// TIA Portal V19 export
FUNCTION "UF" : Void   // FC12, LAD
{ S7_Optimized_Access := 'TRUE' }
// stored: SetENOAutomatically false
   VAR_TEMP   // added for the SCL form of the ladder/FBD networks
      _w1 : Bool;
      _w2 : Bool;
   END_VAR
BEGIN

REGION Network 1: ABFV-201 OPEN F/B
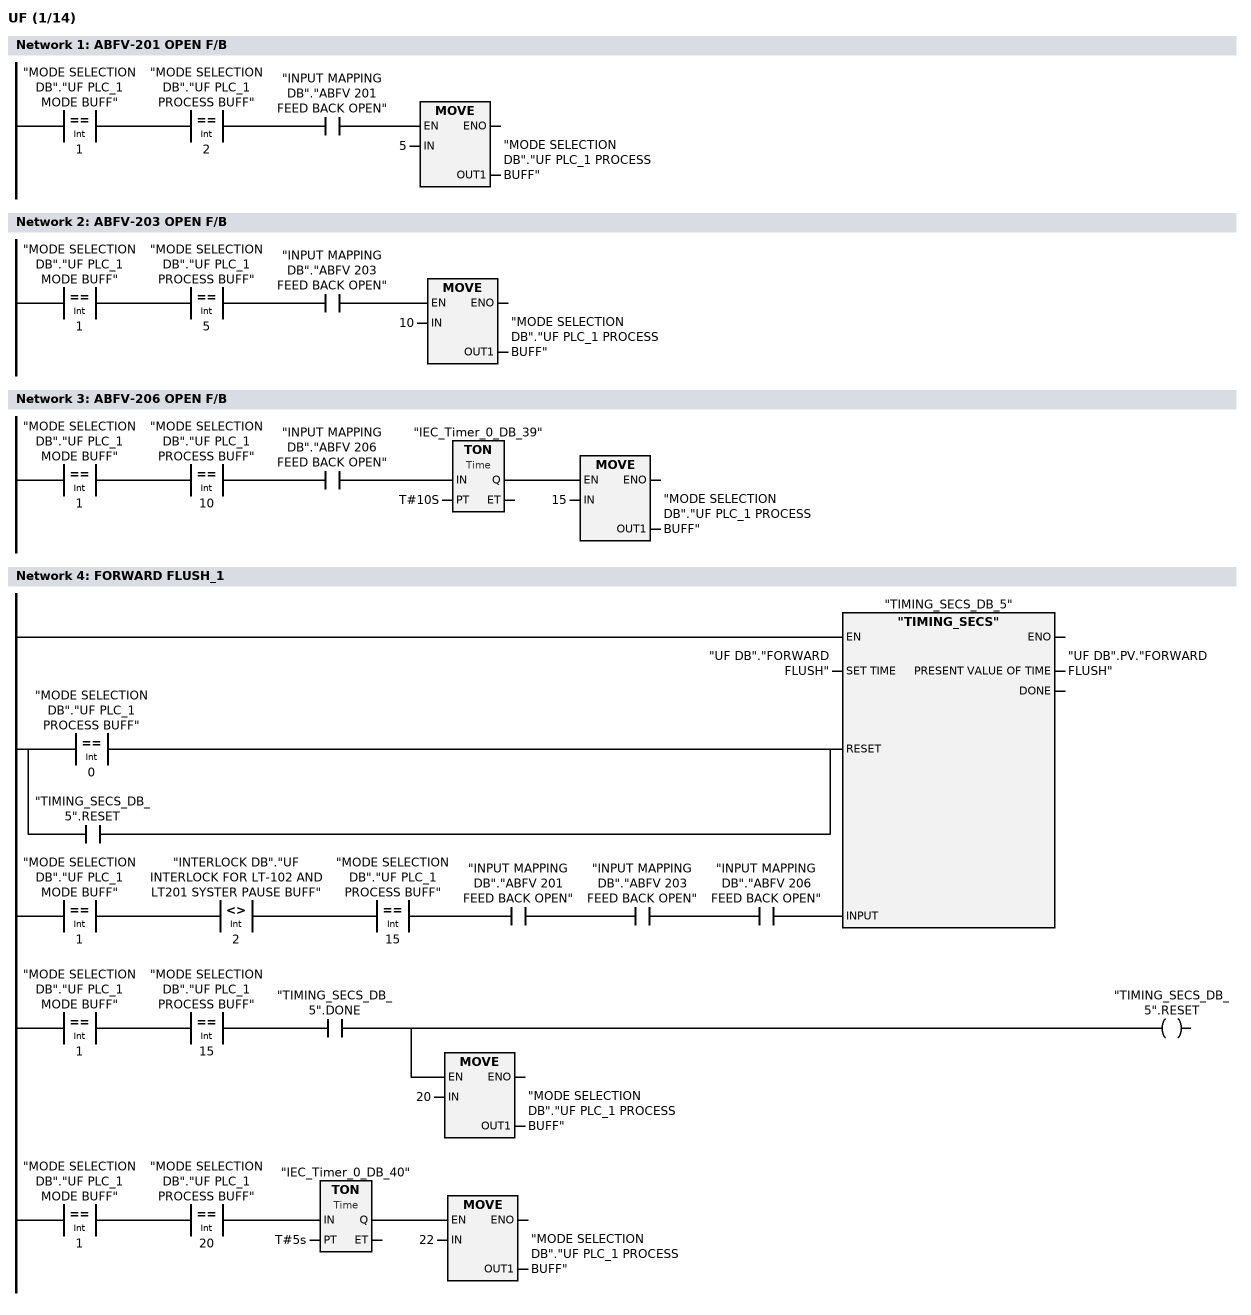
   RUNG wire#powerrail
      { S7_Templates := "SrcType := Int" } EQ_Contact(in1 := "MODE SELECTION DB"."UF PLC_1 MODE BUFF", in2 := 1)
      { S7_Templates := "SrcType := Int" } EQ_Contact(in1 := "MODE SELECTION DB"."UF PLC_1 PROCESS BUFF", in2 := 2)
      Contact( "INPUT MAPPING DB"."ABFV 201 FEED BACK OPEN" )
      Move(in := 5, out1 => "MODE SELECTION DB"."UF PLC_1 PROCESS BUFF")
   END_RUNG
   // the same network as SCL:
   IF ("MODE SELECTION DB"."UF PLC_1 MODE BUFF" = 1) AND ("MODE SELECTION DB"."UF PLC_1 PROCESS BUFF" = 2) AND "INPUT MAPPING DB"."ABFV 201 FEED BACK OPEN" THEN
       "MODE SELECTION DB"."UF PLC_1 PROCESS BUFF" := 5;
   END_IF;
END_REGION

REGION Network 2: ABFV-203 OPEN F/B
   RUNG wire#powerrail
      { S7_Templates := "SrcType := Int" } EQ_Contact(in1 := "MODE SELECTION DB"."UF PLC_1 MODE BUFF", in2 := 1)
      { S7_Templates := "SrcType := Int" } EQ_Contact(in1 := "MODE SELECTION DB"."UF PLC_1 PROCESS BUFF", in2 := 5)
      Contact( "INPUT MAPPING DB"."ABFV 203 FEED BACK OPEN" )
      Move(in := 10, out1 => "MODE SELECTION DB"."UF PLC_1 PROCESS BUFF")
   END_RUNG
   // the same network as SCL:
   IF ("MODE SELECTION DB"."UF PLC_1 MODE BUFF" = 1) AND ("MODE SELECTION DB"."UF PLC_1 PROCESS BUFF" = 5) AND "INPUT MAPPING DB"."ABFV 203 FEED BACK OPEN" THEN
       "MODE SELECTION DB"."UF PLC_1 PROCESS BUFF" := 10;
   END_IF;
END_REGION

REGION Network 3: ABFV-206 OPEN F/B
   RUNG wire#powerrail
      { S7_Templates := "SrcType := Int" } EQ_Contact(in1 := "MODE SELECTION DB"."UF PLC_1 MODE BUFF", in2 := 1)
      { S7_Templates := "SrcType := Int" } EQ_Contact(in1 := "MODE SELECTION DB"."UF PLC_1 PROCESS BUFF", in2 := 10)
      Contact( "INPUT MAPPING DB"."ABFV 206 FEED BACK OPEN" )
      { S7_Templates := "time_type := Time" } "IEC_Timer_0_DB_39".TON(pt := T#10S, et =>)
      Move(in := 15, out1 => "MODE SELECTION DB"."UF PLC_1 PROCESS BUFF")
   END_RUNG
   // the same network as SCL:
   "IEC_Timer_0_DB_39".TON(IN := ("MODE SELECTION DB"."UF PLC_1 MODE BUFF" = 1) AND ("MODE SELECTION DB"."UF PLC_1 PROCESS BUFF" = 10) AND "INPUT MAPPING DB"."ABFV 206 FEED BACK OPEN",
                           PT := T#10S);
   IF "IEC_Timer_0_DB_39".Q THEN "MODE SELECTION DB"."UF PLC_1 PROCESS BUFF" := 15; END_IF;
END_REGION

REGION Network 4: FORWARD FLUSH_1
   RUNG wire#powerrail
      "TIMING_SECS_DB_5"(RESET := wire#w1, INPUT := wire#w2, "SET TIME" := "UF DB"."FORWARD FLUSH", "PRESENT VALUE OF TIME" => "UF DB".PV."FORWARD FLUSH", DONE =>)
   END_RUNG
   RUNG wire#powerrail
      { S7_Templates := "SrcType := Int" } EQ_Contact(in1 := "MODE SELECTION DB"."UF PLC_1 PROCESS BUFF", in2 := 0)
   END_RUNG wire#w1
   RUNG wire#powerrail
      Contact( "TIMING_SECS_DB_5".RESET )
   END_RUNG wire#w1
   RUNG wire#powerrail
      { S7_Templates := "SrcType := Int" } EQ_Contact(in1 := "MODE SELECTION DB"."UF PLC_1 MODE BUFF", in2 := 1)
      { S7_Templates := "SrcType := Int" } NE_Contact(in1 := "INTERLOCK DB"."UF INTERLOCK FOR LT-102 AND LT201 SYSTER PAUSE BUFF", in2 := 2)
      { S7_Templates := "SrcType := Int" } EQ_Contact(in1 := "MODE SELECTION DB"."UF PLC_1 PROCESS BUFF", in2 := 15)
      Contact( "INPUT MAPPING DB"."ABFV 201 FEED BACK OPEN" )
      Contact( "INPUT MAPPING DB"."ABFV 203 FEED BACK OPEN" )
      Contact( "INPUT MAPPING DB"."ABFV 206 FEED BACK OPEN" )
   END_RUNG wire#w2
   RUNG wire#powerrail
      { S7_Templates := "SrcType := Int" } EQ_Contact(in1 := "MODE SELECTION DB"."UF PLC_1 MODE BUFF", in2 := 1)
      { S7_Templates := "SrcType := Int" } EQ_Contact(in1 := "MODE SELECTION DB"."UF PLC_1 PROCESS BUFF", in2 := 15)
      Contact( "TIMING_SECS_DB_5".DONE )
      wire#w3
      Coil( "TIMING_SECS_DB_5".RESET )
   END_RUNG
   RUNG wire#w3
      Move(in := 20, out1 => "MODE SELECTION DB"."UF PLC_1 PROCESS BUFF")
   END_RUNG
   RUNG wire#powerrail
      { S7_Templates := "SrcType := Int" } EQ_Contact(in1 := "MODE SELECTION DB"."UF PLC_1 MODE BUFF", in2 := 1)
      { S7_Templates := "SrcType := Int" } EQ_Contact(in1 := "MODE SELECTION DB"."UF PLC_1 PROCESS BUFF", in2 := 20)
      { S7_Templates := "time_type := Time" } "IEC_Timer_0_DB_40".TON(pt := T#5s, et =>)
      Move(in := 22, out1 => "MODE SELECTION DB"."UF PLC_1 PROCESS BUFF")
   END_RUNG
   // the same network as SCL:
   "TIMING_SECS_DB_5"("SET TIME" := "UF DB"."FORWARD FLUSH",   // "TIMING_SECS"
                      RESET := ("MODE SELECTION DB"."UF PLC_1 PROCESS BUFF" = 0) OR "TIMING_SECS_DB_5".RESET,
                      INPUT := ("MODE SELECTION DB"."UF PLC_1 MODE BUFF" = 1) AND ("INTERLOCK DB"."UF INTERLOCK FOR LT-102 AND LT201 SYSTER PAUSE BUFF" <> 2) AND ("MODE SELECTION DB"."UF PLC_1 PROCESS BUFF" = 15) AND "INPUT MAPPING DB"."ABFV 201 FEED BACK OPEN" AND "INPUT MAPPING DB"."ABFV 203 FEED BACK OPEN" AND "INPUT MAPPING DB"."ABFV 206 FEED BACK OPEN",
                      "PRESENT VALUE OF TIME" => "UF DB".PV."FORWARD FLUSH");
   "TIMING_SECS_DB_5".RESET := ("MODE SELECTION DB"."UF PLC_1 MODE BUFF" = 1) AND ("MODE SELECTION DB"."UF PLC_1 PROCESS BUFF" = 15) AND "TIMING_SECS_DB_5".DONE;
   IF "TIMING_SECS_DB_5".RESET THEN "MODE SELECTION DB"."UF PLC_1 PROCESS BUFF" := 20; END_IF;
   "IEC_Timer_0_DB_40".TON(IN := ("MODE SELECTION DB"."UF PLC_1 MODE BUFF" = 1) AND ("MODE SELECTION DB"."UF PLC_1 PROCESS BUFF" = 20),
                           PT := T#5s);
   IF "IEC_Timer_0_DB_40".Q THEN "MODE SELECTION DB"."UF PLC_1 PROCESS BUFF" := 22; END_IF;
END_REGION

REGION Network 5: OPEN ALL VALVE NEXT PROCESS
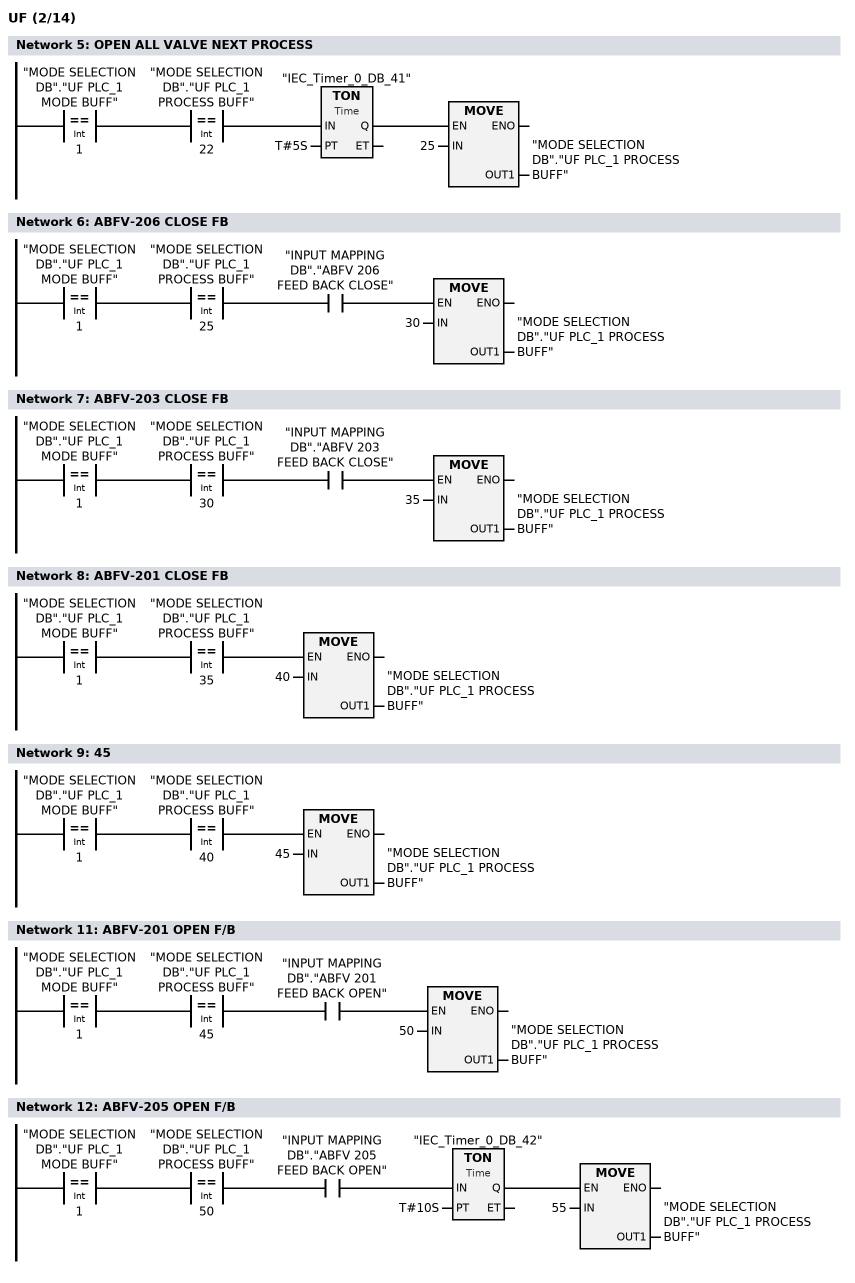
   RUNG wire#powerrail
      { S7_Templates := "SrcType := Int" } EQ_Contact(in1 := "MODE SELECTION DB"."UF PLC_1 MODE BUFF", in2 := 1)
      { S7_Templates := "SrcType := Int" } EQ_Contact(in1 := "MODE SELECTION DB"."UF PLC_1 PROCESS BUFF", in2 := 22)
      { S7_Templates := "time_type := Time" } "IEC_Timer_0_DB_41".TON(pt := T#5S, et =>)
      Move(in := 25, out1 => "MODE SELECTION DB"."UF PLC_1 PROCESS BUFF")
   END_RUNG
   // the same network as SCL:
   "IEC_Timer_0_DB_41".TON(IN := ("MODE SELECTION DB"."UF PLC_1 MODE BUFF" = 1) AND ("MODE SELECTION DB"."UF PLC_1 PROCESS BUFF" = 22),
                           PT := T#5S);
   IF "IEC_Timer_0_DB_41".Q THEN "MODE SELECTION DB"."UF PLC_1 PROCESS BUFF" := 25; END_IF;
END_REGION

REGION Network 6: ABFV-206 CLOSE FB
   RUNG wire#powerrail
      { S7_Templates := "SrcType := Int" } EQ_Contact(in1 := "MODE SELECTION DB"."UF PLC_1 MODE BUFF", in2 := 1)
      { S7_Templates := "SrcType := Int" } EQ_Contact(in1 := "MODE SELECTION DB"."UF PLC_1 PROCESS BUFF", in2 := 25)
      Contact( "INPUT MAPPING DB"."ABFV 206 FEED BACK CLOSE" )
      Move(in := 30, out1 => "MODE SELECTION DB"."UF PLC_1 PROCESS BUFF")
   END_RUNG
   // the same network as SCL:
   IF ("MODE SELECTION DB"."UF PLC_1 MODE BUFF" = 1) AND ("MODE SELECTION DB"."UF PLC_1 PROCESS BUFF" = 25) AND "INPUT MAPPING DB"."ABFV 206 FEED BACK CLOSE" THEN
       "MODE SELECTION DB"."UF PLC_1 PROCESS BUFF" := 30;
   END_IF;
END_REGION

REGION Network 7: ABFV-203 CLOSE FB
   RUNG wire#powerrail
      { S7_Templates := "SrcType := Int" } EQ_Contact(in1 := "MODE SELECTION DB"."UF PLC_1 MODE BUFF", in2 := 1)
      { S7_Templates := "SrcType := Int" } EQ_Contact(in1 := "MODE SELECTION DB"."UF PLC_1 PROCESS BUFF", in2 := 30)
      Contact( "INPUT MAPPING DB"."ABFV 203 FEED BACK CLOSE" )
      Move(in := 35, out1 => "MODE SELECTION DB"."UF PLC_1 PROCESS BUFF")
   END_RUNG
   // the same network as SCL:
   IF ("MODE SELECTION DB"."UF PLC_1 MODE BUFF" = 1) AND ("MODE SELECTION DB"."UF PLC_1 PROCESS BUFF" = 30) AND "INPUT MAPPING DB"."ABFV 203 FEED BACK CLOSE" THEN
       "MODE SELECTION DB"."UF PLC_1 PROCESS BUFF" := 35;
   END_IF;
END_REGION

REGION Network 8: ABFV-201 CLOSE FB
   RUNG wire#powerrail
      { S7_Templates := "SrcType := Int" } EQ_Contact(in1 := "MODE SELECTION DB"."UF PLC_1 MODE BUFF", in2 := 1)
      { S7_Templates := "SrcType := Int" } EQ_Contact(in1 := "MODE SELECTION DB"."UF PLC_1 PROCESS BUFF", in2 := 35)
      Move(in := 40, out1 => "MODE SELECTION DB"."UF PLC_1 PROCESS BUFF")
   END_RUNG
   // the same network as SCL:
   IF ("MODE SELECTION DB"."UF PLC_1 MODE BUFF" = 1) AND ("MODE SELECTION DB"."UF PLC_1 PROCESS BUFF" = 35) THEN
       "MODE SELECTION DB"."UF PLC_1 PROCESS BUFF" := 40;
   END_IF;
END_REGION

REGION Network 9: 45
   RUNG wire#powerrail
      { S7_Templates := "SrcType := Int" } EQ_Contact(in1 := "MODE SELECTION DB"."UF PLC_1 MODE BUFF", in2 := 1)
      { S7_Templates := "SrcType := Int" } EQ_Contact(in1 := "MODE SELECTION DB"."UF PLC_1 PROCESS BUFF", in2 := 40)
      Move(in := 45, out1 => "MODE SELECTION DB"."UF PLC_1 PROCESS BUFF")
   END_RUNG
   // the same network as SCL:
   IF ("MODE SELECTION DB"."UF PLC_1 MODE BUFF" = 1) AND ("MODE SELECTION DB"."UF PLC_1 PROCESS BUFF" = 40) THEN
       "MODE SELECTION DB"."UF PLC_1 PROCESS BUFF" := 45;
   END_IF;
END_REGION

REGION Network 11: ABFV-201 OPEN F/B
   RUNG wire#powerrail
      { S7_Templates := "SrcType := Int" } EQ_Contact(in1 := "MODE SELECTION DB"."UF PLC_1 MODE BUFF", in2 := 1)
      { S7_Templates := "SrcType := Int" } EQ_Contact(in1 := "MODE SELECTION DB"."UF PLC_1 PROCESS BUFF", in2 := 45)
      Contact( "INPUT MAPPING DB"."ABFV 201 FEED BACK OPEN" )
      Move(in := 50, out1 => "MODE SELECTION DB"."UF PLC_1 PROCESS BUFF")
   END_RUNG
   // the same network as SCL:
   IF ("MODE SELECTION DB"."UF PLC_1 MODE BUFF" = 1) AND ("MODE SELECTION DB"."UF PLC_1 PROCESS BUFF" = 45) AND "INPUT MAPPING DB"."ABFV 201 FEED BACK OPEN" THEN
       "MODE SELECTION DB"."UF PLC_1 PROCESS BUFF" := 50;
   END_IF;
END_REGION

REGION Network 12: ABFV-205 OPEN F/B
   RUNG wire#powerrail
      { S7_Templates := "SrcType := Int" } EQ_Contact(in1 := "MODE SELECTION DB"."UF PLC_1 MODE BUFF", in2 := 1)
      { S7_Templates := "SrcType := Int" } EQ_Contact(in1 := "MODE SELECTION DB"."UF PLC_1 PROCESS BUFF", in2 := 50)
      Contact( "INPUT MAPPING DB"."ABFV 205 FEED BACK OPEN" )
      { S7_Templates := "time_type := Time" } "IEC_Timer_0_DB_42".TON(pt := T#10S, et =>)
      Move(in := 55, out1 => "MODE SELECTION DB"."UF PLC_1 PROCESS BUFF")
   END_RUNG
   // the same network as SCL:
   "IEC_Timer_0_DB_42".TON(IN := ("MODE SELECTION DB"."UF PLC_1 MODE BUFF" = 1) AND ("MODE SELECTION DB"."UF PLC_1 PROCESS BUFF" = 50) AND "INPUT MAPPING DB"."ABFV 205 FEED BACK OPEN",
                           PT := T#10S);
   IF "IEC_Timer_0_DB_42".Q THEN "MODE SELECTION DB"."UF PLC_1 PROCESS BUFF" := 55; END_IF;
END_REGION

REGION Network 13: FILTRATION MODE
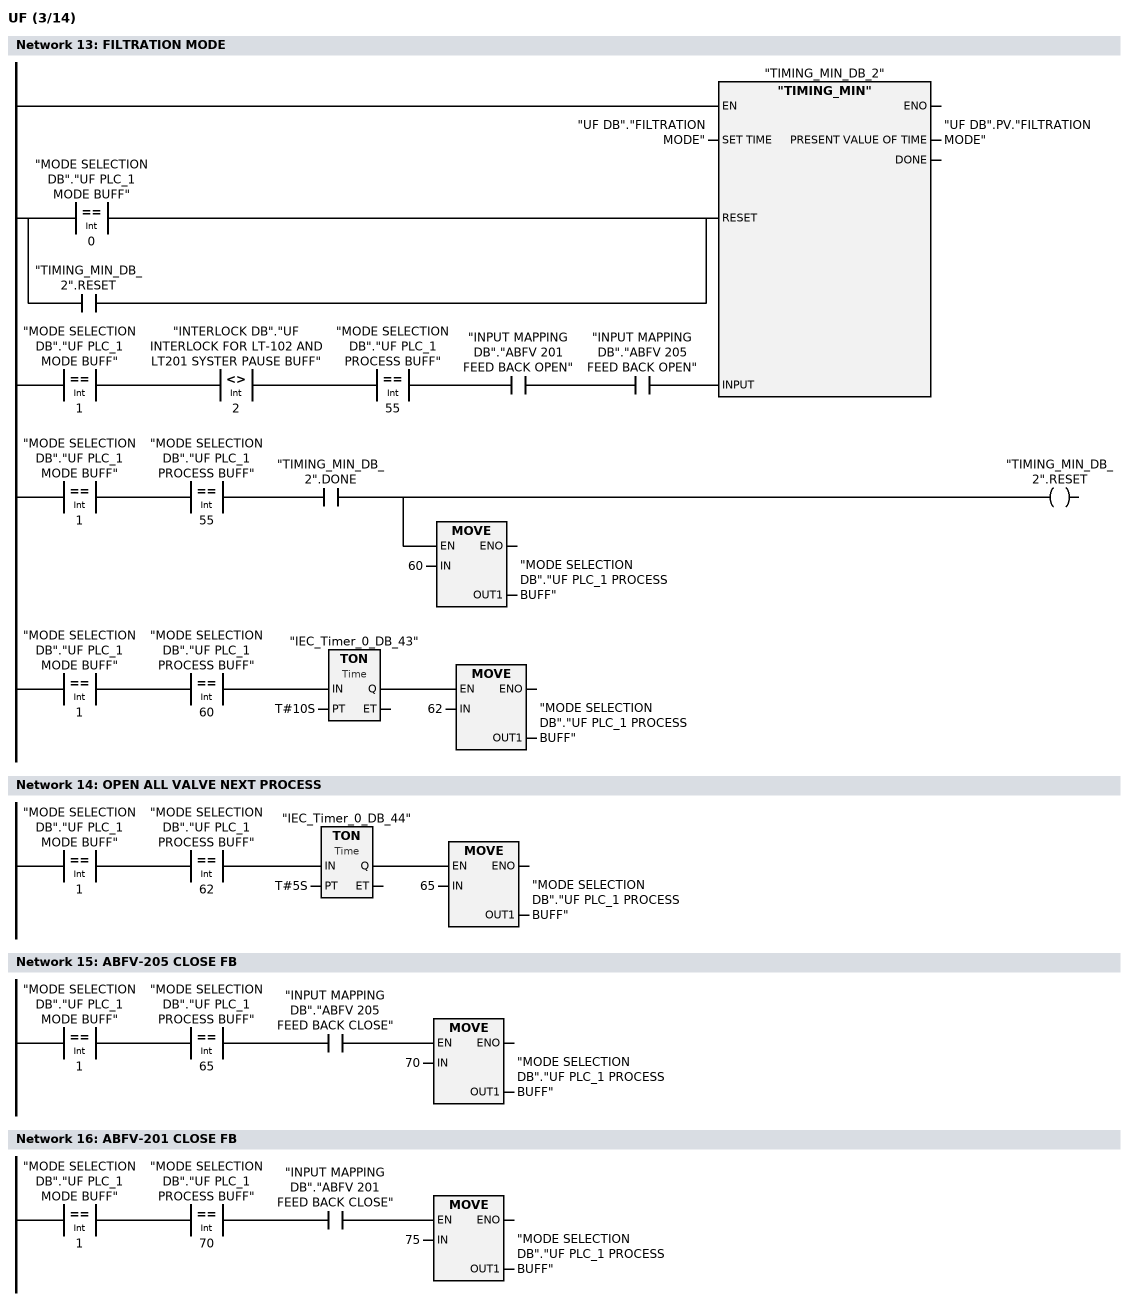
   RUNG wire#powerrail
      "TIMING_MIN_DB_2"(RESET := wire#w1, INPUT := wire#w2, "SET TIME" := "UF DB"."FILTRATION MODE", "PRESENT VALUE OF TIME" => "UF DB".PV."FILTRATION MODE", DONE =>)
   END_RUNG
   RUNG wire#powerrail
      { S7_Templates := "SrcType := Int" } EQ_Contact(in1 := "MODE SELECTION DB"."UF PLC_1 MODE BUFF", in2 := 0)
   END_RUNG wire#w1
   RUNG wire#powerrail
      Contact( "TIMING_MIN_DB_2".RESET )
   END_RUNG wire#w1
   RUNG wire#powerrail
      { S7_Templates := "SrcType := Int" } EQ_Contact(in1 := "MODE SELECTION DB"."UF PLC_1 MODE BUFF", in2 := 1)
      { S7_Templates := "SrcType := Int" } NE_Contact(in1 := "INTERLOCK DB"."UF INTERLOCK FOR LT-102 AND LT201 SYSTER PAUSE BUFF", in2 := 2)
      { S7_Templates := "SrcType := Int" } EQ_Contact(in1 := "MODE SELECTION DB"."UF PLC_1 PROCESS BUFF", in2 := 55)
      Contact( "INPUT MAPPING DB"."ABFV 201 FEED BACK OPEN" )
      Contact( "INPUT MAPPING DB"."ABFV 205 FEED BACK OPEN" )
   END_RUNG wire#w2
   RUNG wire#powerrail
      { S7_Templates := "SrcType := Int" } EQ_Contact(in1 := "MODE SELECTION DB"."UF PLC_1 MODE BUFF", in2 := 1)
      { S7_Templates := "SrcType := Int" } EQ_Contact(in1 := "MODE SELECTION DB"."UF PLC_1 PROCESS BUFF", in2 := 55)
      Contact( "TIMING_MIN_DB_2".DONE )
      wire#w3
      Coil( "TIMING_MIN_DB_2".RESET )
   END_RUNG
   RUNG wire#w3
      Move(in := 60, out1 => "MODE SELECTION DB"."UF PLC_1 PROCESS BUFF")
   END_RUNG
   RUNG wire#powerrail
      { S7_Templates := "SrcType := Int" } EQ_Contact(in1 := "MODE SELECTION DB"."UF PLC_1 MODE BUFF", in2 := 1)
      { S7_Templates := "SrcType := Int" } EQ_Contact(in1 := "MODE SELECTION DB"."UF PLC_1 PROCESS BUFF", in2 := 60)
      { S7_Templates := "time_type := Time" } "IEC_Timer_0_DB_43".TON(pt := T#10S, et =>)
      Move(in := 62, out1 => "MODE SELECTION DB"."UF PLC_1 PROCESS BUFF")
   END_RUNG
   // the same network as SCL:
   "TIMING_MIN_DB_2"("SET TIME" := "UF DB"."FILTRATION MODE",   // "TIMING_MIN"
                     RESET := ("MODE SELECTION DB"."UF PLC_1 MODE BUFF" = 0) OR "TIMING_MIN_DB_2".RESET,
                     INPUT := ("MODE SELECTION DB"."UF PLC_1 MODE BUFF" = 1) AND ("INTERLOCK DB"."UF INTERLOCK FOR LT-102 AND LT201 SYSTER PAUSE BUFF" <> 2) AND ("MODE SELECTION DB"."UF PLC_1 PROCESS BUFF" = 55) AND "INPUT MAPPING DB"."ABFV 201 FEED BACK OPEN" AND "INPUT MAPPING DB"."ABFV 205 FEED BACK OPEN",
                     "PRESENT VALUE OF TIME" => "UF DB".PV."FILTRATION MODE");
   "TIMING_MIN_DB_2".RESET := ("MODE SELECTION DB"."UF PLC_1 MODE BUFF" = 1) AND ("MODE SELECTION DB"."UF PLC_1 PROCESS BUFF" = 55) AND "TIMING_MIN_DB_2".DONE;
   IF "TIMING_MIN_DB_2".RESET THEN "MODE SELECTION DB"."UF PLC_1 PROCESS BUFF" := 60; END_IF;
   "IEC_Timer_0_DB_43".TON(IN := ("MODE SELECTION DB"."UF PLC_1 MODE BUFF" = 1) AND ("MODE SELECTION DB"."UF PLC_1 PROCESS BUFF" = 60),
                           PT := T#10S);
   IF "IEC_Timer_0_DB_43".Q THEN "MODE SELECTION DB"."UF PLC_1 PROCESS BUFF" := 62; END_IF;
END_REGION

REGION Network 14: OPEN ALL VALVE NEXT PROCESS
   RUNG wire#powerrail
      { S7_Templates := "SrcType := Int" } EQ_Contact(in1 := "MODE SELECTION DB"."UF PLC_1 MODE BUFF", in2 := 1)
      { S7_Templates := "SrcType := Int" } EQ_Contact(in1 := "MODE SELECTION DB"."UF PLC_1 PROCESS BUFF", in2 := 62)
      { S7_Templates := "time_type := Time" } "IEC_Timer_0_DB_44".TON(pt := T#5S, et =>)
      Move(in := 65, out1 => "MODE SELECTION DB"."UF PLC_1 PROCESS BUFF")
   END_RUNG
   // the same network as SCL:
   "IEC_Timer_0_DB_44".TON(IN := ("MODE SELECTION DB"."UF PLC_1 MODE BUFF" = 1) AND ("MODE SELECTION DB"."UF PLC_1 PROCESS BUFF" = 62),
                           PT := T#5S);
   IF "IEC_Timer_0_DB_44".Q THEN "MODE SELECTION DB"."UF PLC_1 PROCESS BUFF" := 65; END_IF;
END_REGION

REGION Network 15: ABFV-205 CLOSE FB
   RUNG wire#powerrail
      { S7_Templates := "SrcType := Int" } EQ_Contact(in1 := "MODE SELECTION DB"."UF PLC_1 MODE BUFF", in2 := 1)
      { S7_Templates := "SrcType := Int" } EQ_Contact(in1 := "MODE SELECTION DB"."UF PLC_1 PROCESS BUFF", in2 := 65)
      Contact( "INPUT MAPPING DB"."ABFV 205 FEED BACK CLOSE" )
      Move(in := 70, out1 => "MODE SELECTION DB"."UF PLC_1 PROCESS BUFF")
   END_RUNG
   // the same network as SCL:
   IF ("MODE SELECTION DB"."UF PLC_1 MODE BUFF" = 1) AND ("MODE SELECTION DB"."UF PLC_1 PROCESS BUFF" = 65) AND "INPUT MAPPING DB"."ABFV 205 FEED BACK CLOSE" THEN
       "MODE SELECTION DB"."UF PLC_1 PROCESS BUFF" := 70;
   END_IF;
END_REGION

REGION Network 16: ABFV-201 CLOSE FB
   RUNG wire#powerrail
      { S7_Templates := "SrcType := Int" } EQ_Contact(in1 := "MODE SELECTION DB"."UF PLC_1 MODE BUFF", in2 := 1)
      { S7_Templates := "SrcType := Int" } EQ_Contact(in1 := "MODE SELECTION DB"."UF PLC_1 PROCESS BUFF", in2 := 70)
      Contact( "INPUT MAPPING DB"."ABFV 201 FEED BACK CLOSE" )
      Move(in := 75, out1 => "MODE SELECTION DB"."UF PLC_1 PROCESS BUFF")
   END_RUNG
   // the same network as SCL:
   IF ("MODE SELECTION DB"."UF PLC_1 MODE BUFF" = 1) AND ("MODE SELECTION DB"."UF PLC_1 PROCESS BUFF" = 70) AND "INPUT MAPPING DB"."ABFV 201 FEED BACK CLOSE" THEN
       "MODE SELECTION DB"."UF PLC_1 PROCESS BUFF" := 75;
   END_IF;
END_REGION

REGION Network 17: 80
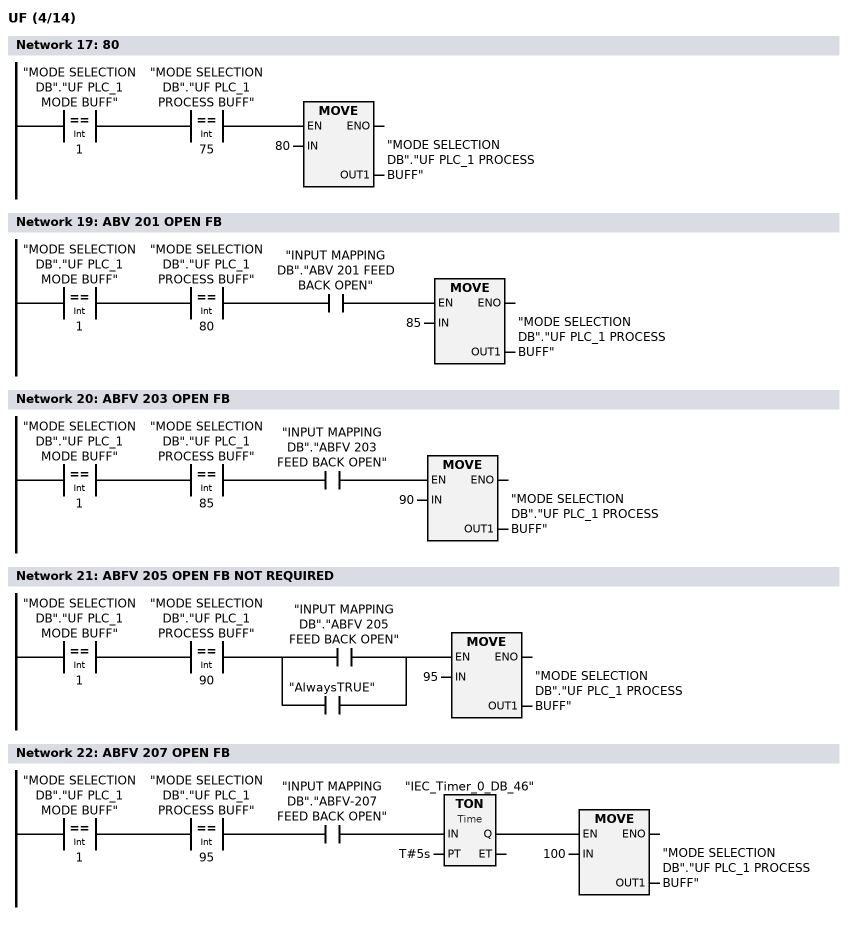
   RUNG wire#powerrail
      { S7_Templates := "SrcType := Int" } EQ_Contact(in1 := "MODE SELECTION DB"."UF PLC_1 MODE BUFF", in2 := 1)
      { S7_Templates := "SrcType := Int" } EQ_Contact(in1 := "MODE SELECTION DB"."UF PLC_1 PROCESS BUFF", in2 := 75)
      Move(in := 80, out1 => "MODE SELECTION DB"."UF PLC_1 PROCESS BUFF")
   END_RUNG
   // the same network as SCL:
   IF ("MODE SELECTION DB"."UF PLC_1 MODE BUFF" = 1) AND ("MODE SELECTION DB"."UF PLC_1 PROCESS BUFF" = 75) THEN
       "MODE SELECTION DB"."UF PLC_1 PROCESS BUFF" := 80;
   END_IF;
END_REGION

REGION Network 19: ABV 201 OPEN FB
   RUNG wire#powerrail
      { S7_Templates := "SrcType := Int" } EQ_Contact(in1 := "MODE SELECTION DB"."UF PLC_1 MODE BUFF", in2 := 1)
      { S7_Templates := "SrcType := Int" } EQ_Contact(in1 := "MODE SELECTION DB"."UF PLC_1 PROCESS BUFF", in2 := 80)
      Contact( "INPUT MAPPING DB"."ABV 201 FEED BACK OPEN" )
      Move(in := 85, out1 => "MODE SELECTION DB"."UF PLC_1 PROCESS BUFF")
   END_RUNG
   // the same network as SCL:
   IF ("MODE SELECTION DB"."UF PLC_1 MODE BUFF" = 1) AND ("MODE SELECTION DB"."UF PLC_1 PROCESS BUFF" = 80) AND "INPUT MAPPING DB"."ABV 201 FEED BACK OPEN" THEN
       "MODE SELECTION DB"."UF PLC_1 PROCESS BUFF" := 85;
   END_IF;
END_REGION

REGION Network 20: ABFV 203 OPEN FB
   RUNG wire#powerrail
      { S7_Templates := "SrcType := Int" } EQ_Contact(in1 := "MODE SELECTION DB"."UF PLC_1 MODE BUFF", in2 := 1)
      { S7_Templates := "SrcType := Int" } EQ_Contact(in1 := "MODE SELECTION DB"."UF PLC_1 PROCESS BUFF", in2 := 85)
      Contact( "INPUT MAPPING DB"."ABFV 203 FEED BACK OPEN" )
      Move(in := 90, out1 => "MODE SELECTION DB"."UF PLC_1 PROCESS BUFF")
   END_RUNG
   // the same network as SCL:
   IF ("MODE SELECTION DB"."UF PLC_1 MODE BUFF" = 1) AND ("MODE SELECTION DB"."UF PLC_1 PROCESS BUFF" = 85) AND "INPUT MAPPING DB"."ABFV 203 FEED BACK OPEN" THEN
       "MODE SELECTION DB"."UF PLC_1 PROCESS BUFF" := 90;
   END_IF;
END_REGION

REGION Network 21: ABFV 205 OPEN FB NOT REQUIRED
   RUNG wire#powerrail
      { S7_Templates := "SrcType := Int" } EQ_Contact(in1 := "MODE SELECTION DB"."UF PLC_1 MODE BUFF", in2 := 1)
      { S7_Templates := "SrcType := Int" } EQ_Contact(in1 := "MODE SELECTION DB"."UF PLC_1 PROCESS BUFF", in2 := 90)
      wire#w1
      Contact( "INPUT MAPPING DB"."ABFV 205 FEED BACK OPEN" )
      wire#w2
      Move(in := 95, out1 => "MODE SELECTION DB"."UF PLC_1 PROCESS BUFF")
   END_RUNG
   RUNG wire#w1
      Contact( "AlwaysTRUE" )
   END_RUNG wire#w2
   // the same network as SCL:
   IF ("MODE SELECTION DB"."UF PLC_1 MODE BUFF" = 1) AND ("MODE SELECTION DB"."UF PLC_1 PROCESS BUFF" = 90) AND ("INPUT MAPPING DB"."ABFV 205 FEED BACK OPEN" OR "AlwaysTRUE") THEN
       "MODE SELECTION DB"."UF PLC_1 PROCESS BUFF" := 95;
   END_IF;
END_REGION

REGION Network 22: ABFV 207 OPEN FB
   RUNG wire#powerrail
      { S7_Templates := "SrcType := Int" } EQ_Contact(in1 := "MODE SELECTION DB"."UF PLC_1 MODE BUFF", in2 := 1)
      { S7_Templates := "SrcType := Int" } EQ_Contact(in1 := "MODE SELECTION DB"."UF PLC_1 PROCESS BUFF", in2 := 95)
      Contact( "INPUT MAPPING DB"."ABFV-207 FEED BACK OPEN" )
      { S7_Templates := "time_type := Time" } "IEC_Timer_0_DB_46".TON(pt := T#5s, et =>)
      Move(in := 100, out1 => "MODE SELECTION DB"."UF PLC_1 PROCESS BUFF")
   END_RUNG
   // the same network as SCL:
   "IEC_Timer_0_DB_46".TON(IN := ("MODE SELECTION DB"."UF PLC_1 MODE BUFF" = 1) AND ("MODE SELECTION DB"."UF PLC_1 PROCESS BUFF" = 95) AND "INPUT MAPPING DB"."ABFV-207 FEED BACK OPEN",
                           PT := T#5s);
   IF "IEC_Timer_0_DB_46".Q THEN "MODE SELECTION DB"."UF PLC_1 PROCESS BUFF" := 100; END_IF;
END_REGION

REGION Network 23: AIR INLET
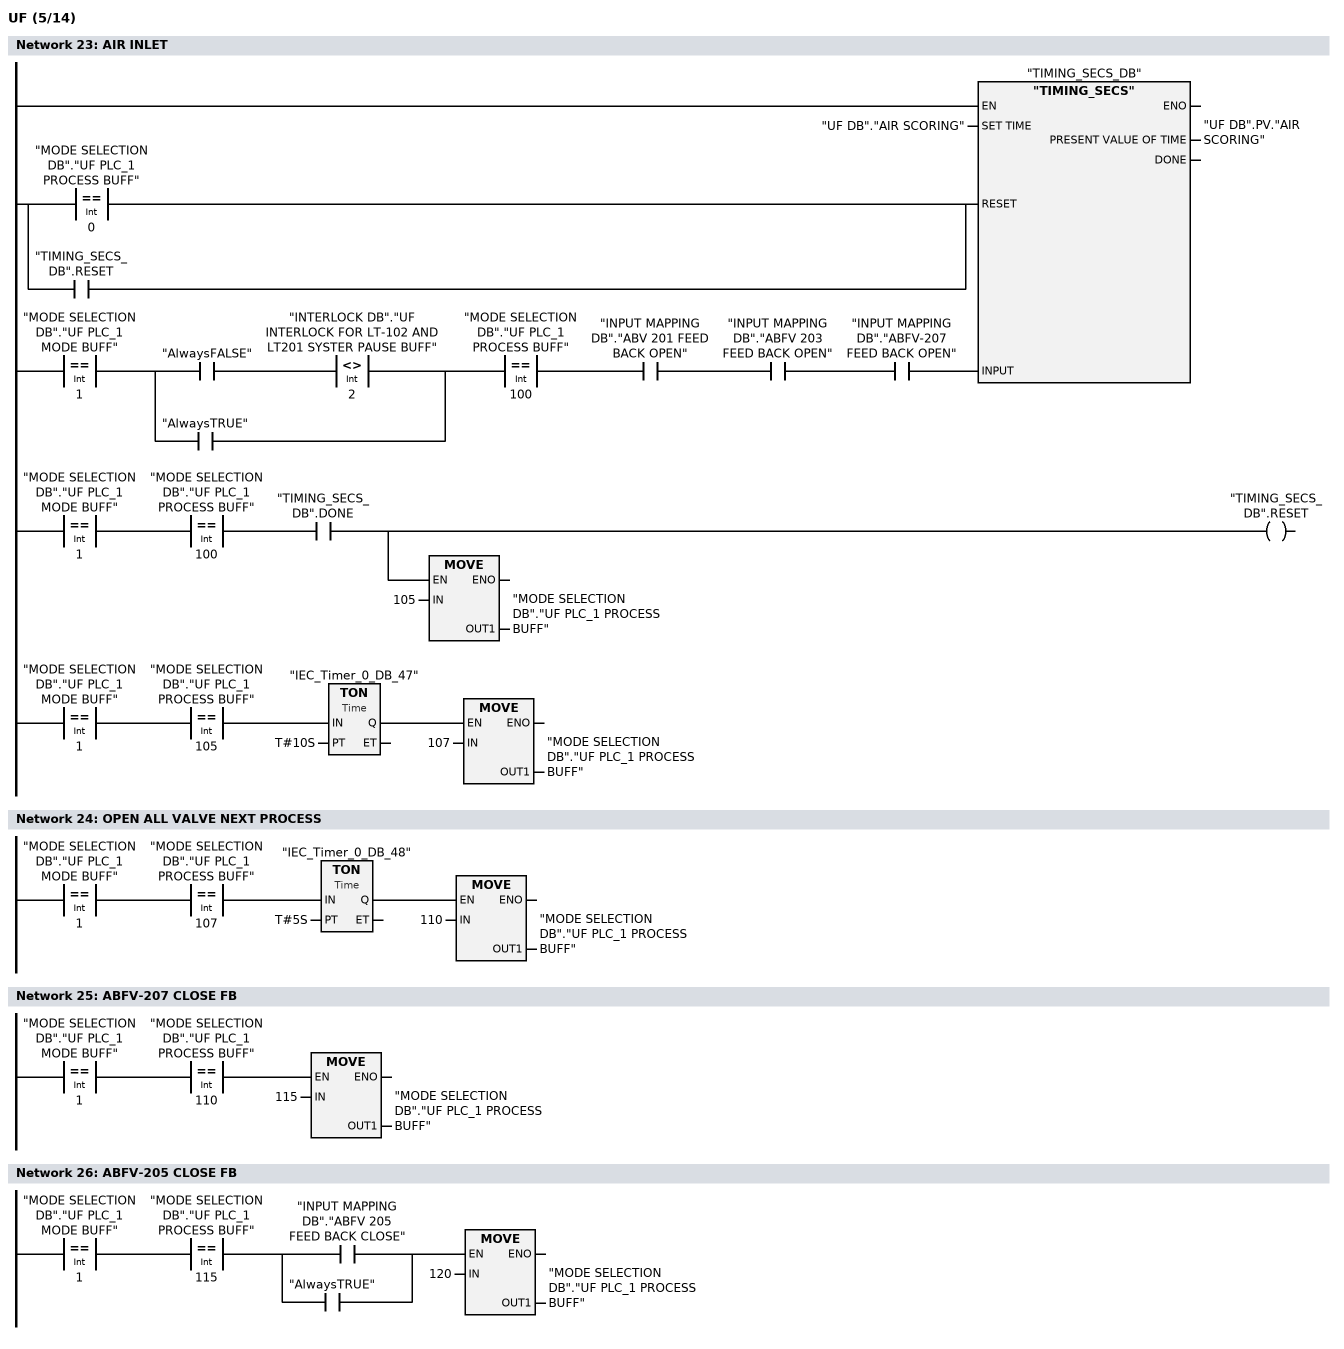
   RUNG wire#powerrail
      "TIMING_SECS_DB"(RESET := wire#w1, INPUT := wire#w4, "SET TIME" := "UF DB"."AIR SCORING", "PRESENT VALUE OF TIME" => "UF DB".PV."AIR SCORING", DONE =>)
   END_RUNG
   RUNG wire#powerrail
      { S7_Templates := "SrcType := Int" } EQ_Contact(in1 := "MODE SELECTION DB"."UF PLC_1 PROCESS BUFF", in2 := 0)
   END_RUNG wire#w1
   RUNG wire#powerrail
      Contact( "TIMING_SECS_DB".RESET )
   END_RUNG wire#w1
   RUNG wire#powerrail
      { S7_Templates := "SrcType := Int" } EQ_Contact(in1 := "MODE SELECTION DB"."UF PLC_1 MODE BUFF", in2 := 1)
      wire#w2
      Contact( "AlwaysFALSE" )
      { S7_Templates := "SrcType := Int" } NE_Contact(in1 := "INTERLOCK DB"."UF INTERLOCK FOR LT-102 AND LT201 SYSTER PAUSE BUFF", in2 := 2)
      wire#w3
      { S7_Templates := "SrcType := Int" } EQ_Contact(in1 := "MODE SELECTION DB"."UF PLC_1 PROCESS BUFF", in2 := 100)
      Contact( "INPUT MAPPING DB"."ABV 201 FEED BACK OPEN" )
      Contact( "INPUT MAPPING DB"."ABFV 203 FEED BACK OPEN" )
      Contact( "INPUT MAPPING DB"."ABFV-207 FEED BACK OPEN" )
   END_RUNG wire#w4
   RUNG wire#w2
      Contact( "AlwaysTRUE" )
   END_RUNG wire#w3
   RUNG wire#powerrail
      { S7_Templates := "SrcType := Int" } EQ_Contact(in1 := "MODE SELECTION DB"."UF PLC_1 MODE BUFF", in2 := 1)
      { S7_Templates := "SrcType := Int" } EQ_Contact(in1 := "MODE SELECTION DB"."UF PLC_1 PROCESS BUFF", in2 := 100)
      Contact( "TIMING_SECS_DB".DONE )
      wire#w5
      Coil( "TIMING_SECS_DB".RESET )
   END_RUNG
   RUNG wire#w5
      Move(in := 105, out1 => "MODE SELECTION DB"."UF PLC_1 PROCESS BUFF")
   END_RUNG
   RUNG wire#powerrail
      { S7_Templates := "SrcType := Int" } EQ_Contact(in1 := "MODE SELECTION DB"."UF PLC_1 MODE BUFF", in2 := 1)
      { S7_Templates := "SrcType := Int" } EQ_Contact(in1 := "MODE SELECTION DB"."UF PLC_1 PROCESS BUFF", in2 := 105)
      { S7_Templates := "time_type := Time" } "IEC_Timer_0_DB_47".TON(pt := T#10S, et =>)
      Move(in := 107, out1 => "MODE SELECTION DB"."UF PLC_1 PROCESS BUFF")
   END_RUNG
   // the same network as SCL:
   "TIMING_SECS_DB"("SET TIME" := "UF DB"."AIR SCORING",   // "TIMING_SECS"
                    RESET := ("MODE SELECTION DB"."UF PLC_1 PROCESS BUFF" = 0) OR "TIMING_SECS_DB".RESET,
                    INPUT := ("MODE SELECTION DB"."UF PLC_1 MODE BUFF" = 1) AND (("AlwaysFALSE" AND ("INTERLOCK DB"."UF INTERLOCK FOR LT-102 AND LT201 SYSTER PAUSE BUFF" <> 2)) OR "AlwaysTRUE") AND ("MODE SELECTION DB"."UF PLC_1 PROCESS BUFF" = 100) AND "INPUT MAPPING DB"."ABV 201 FEED BACK OPEN" AND "INPUT MAPPING DB"."ABFV 203 FEED BACK OPEN" AND "INPUT MAPPING DB"."ABFV-207 FEED BACK OPEN",
                    "PRESENT VALUE OF TIME" => "UF DB".PV."AIR SCORING");
   "TIMING_SECS_DB".RESET := ("MODE SELECTION DB"."UF PLC_1 MODE BUFF" = 1) AND ("MODE SELECTION DB"."UF PLC_1 PROCESS BUFF" = 100) AND "TIMING_SECS_DB".DONE;
   IF "TIMING_SECS_DB".RESET THEN "MODE SELECTION DB"."UF PLC_1 PROCESS BUFF" := 105; END_IF;
   "IEC_Timer_0_DB_47".TON(IN := ("MODE SELECTION DB"."UF PLC_1 MODE BUFF" = 1) AND ("MODE SELECTION DB"."UF PLC_1 PROCESS BUFF" = 105),
                           PT := T#10S);
   IF "IEC_Timer_0_DB_47".Q THEN "MODE SELECTION DB"."UF PLC_1 PROCESS BUFF" := 107; END_IF;
END_REGION

REGION Network 24: OPEN ALL VALVE NEXT PROCESS
   RUNG wire#powerrail
      { S7_Templates := "SrcType := Int" } EQ_Contact(in1 := "MODE SELECTION DB"."UF PLC_1 MODE BUFF", in2 := 1)
      { S7_Templates := "SrcType := Int" } EQ_Contact(in1 := "MODE SELECTION DB"."UF PLC_1 PROCESS BUFF", in2 := 107)
      { S7_Templates := "time_type := Time" } "IEC_Timer_0_DB_48".TON(pt := T#5S, et =>)
      Move(in := 110, out1 => "MODE SELECTION DB"."UF PLC_1 PROCESS BUFF")
   END_RUNG
   // the same network as SCL:
   "IEC_Timer_0_DB_48".TON(IN := ("MODE SELECTION DB"."UF PLC_1 MODE BUFF" = 1) AND ("MODE SELECTION DB"."UF PLC_1 PROCESS BUFF" = 107),
                           PT := T#5S);
   IF "IEC_Timer_0_DB_48".Q THEN "MODE SELECTION DB"."UF PLC_1 PROCESS BUFF" := 110; END_IF;
END_REGION

REGION Network 25: ABFV-207 CLOSE FB
   RUNG wire#powerrail
      { S7_Templates := "SrcType := Int" } EQ_Contact(in1 := "MODE SELECTION DB"."UF PLC_1 MODE BUFF", in2 := 1)
      { S7_Templates := "SrcType := Int" } EQ_Contact(in1 := "MODE SELECTION DB"."UF PLC_1 PROCESS BUFF", in2 := 110)
      Move(in := 115, out1 => "MODE SELECTION DB"."UF PLC_1 PROCESS BUFF")
   END_RUNG
   // the same network as SCL:
   IF ("MODE SELECTION DB"."UF PLC_1 MODE BUFF" = 1) AND ("MODE SELECTION DB"."UF PLC_1 PROCESS BUFF" = 110) THEN
       "MODE SELECTION DB"."UF PLC_1 PROCESS BUFF" := 115;
   END_IF;
END_REGION

REGION Network 26: ABFV-205 CLOSE FB
   RUNG wire#powerrail
      { S7_Templates := "SrcType := Int" } EQ_Contact(in1 := "MODE SELECTION DB"."UF PLC_1 MODE BUFF", in2 := 1)
      { S7_Templates := "SrcType := Int" } EQ_Contact(in1 := "MODE SELECTION DB"."UF PLC_1 PROCESS BUFF", in2 := 115)
      wire#w1
      Contact( "INPUT MAPPING DB"."ABFV 205 FEED BACK CLOSE" )
      wire#w2
      Move(in := 120, out1 => "MODE SELECTION DB"."UF PLC_1 PROCESS BUFF")
   END_RUNG
   RUNG wire#w1
      Contact( "AlwaysTRUE" )
   END_RUNG wire#w2
   // the same network as SCL:
   IF ("MODE SELECTION DB"."UF PLC_1 MODE BUFF" = 1) AND ("MODE SELECTION DB"."UF PLC_1 PROCESS BUFF" = 115) AND ("INPUT MAPPING DB"."ABFV 205 FEED BACK CLOSE" OR "AlwaysTRUE") THEN
       "MODE SELECTION DB"."UF PLC_1 PROCESS BUFF" := 120;
   END_IF;
END_REGION

REGION Network 27: ABFV-203 CLOSE FB
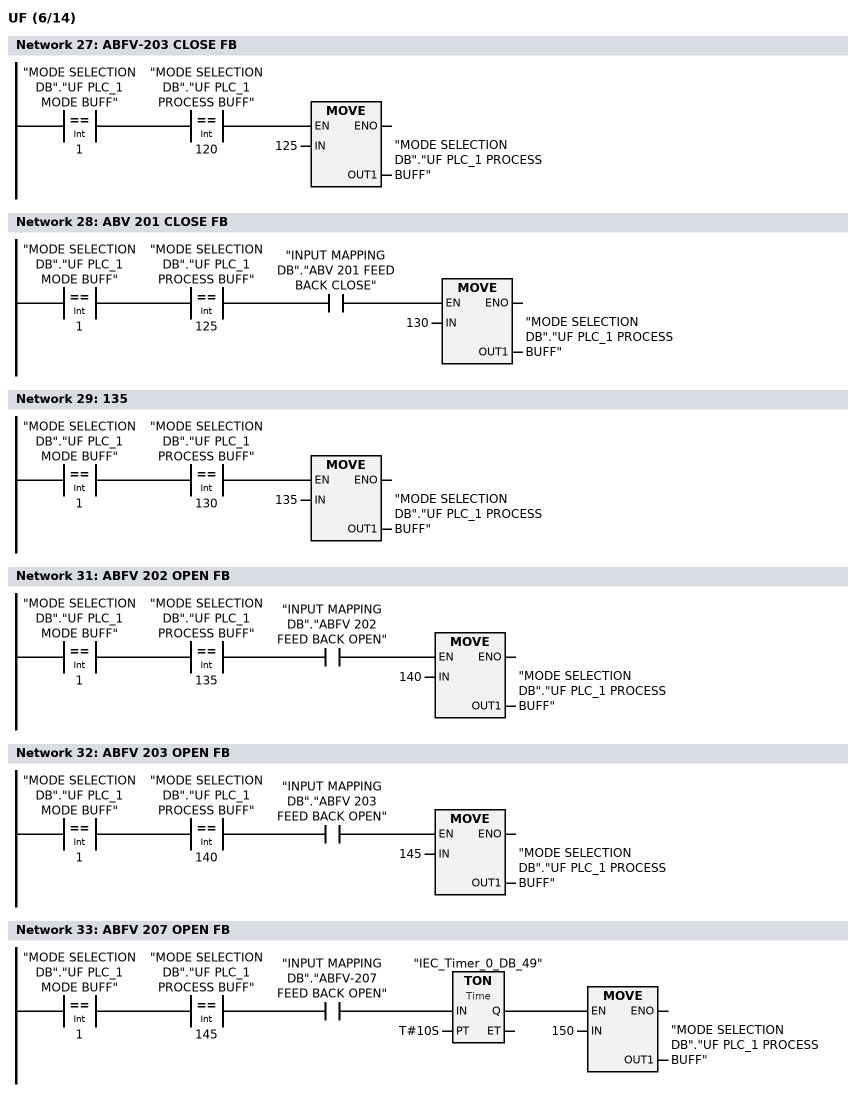
   RUNG wire#powerrail
      { S7_Templates := "SrcType := Int" } EQ_Contact(in1 := "MODE SELECTION DB"."UF PLC_1 MODE BUFF", in2 := 1)
      { S7_Templates := "SrcType := Int" } EQ_Contact(in1 := "MODE SELECTION DB"."UF PLC_1 PROCESS BUFF", in2 := 120)
      Move(in := 125, out1 => "MODE SELECTION DB"."UF PLC_1 PROCESS BUFF")
   END_RUNG
   // the same network as SCL:
   IF ("MODE SELECTION DB"."UF PLC_1 MODE BUFF" = 1) AND ("MODE SELECTION DB"."UF PLC_1 PROCESS BUFF" = 120) THEN
       "MODE SELECTION DB"."UF PLC_1 PROCESS BUFF" := 125;
   END_IF;
END_REGION

REGION Network 28: ABV 201 CLOSE FB
   RUNG wire#powerrail
      { S7_Templates := "SrcType := Int" } EQ_Contact(in1 := "MODE SELECTION DB"."UF PLC_1 MODE BUFF", in2 := 1)
      { S7_Templates := "SrcType := Int" } EQ_Contact(in1 := "MODE SELECTION DB"."UF PLC_1 PROCESS BUFF", in2 := 125)
      Contact( "INPUT MAPPING DB"."ABV 201 FEED BACK CLOSE" )
      Move(in := 130, out1 => "MODE SELECTION DB"."UF PLC_1 PROCESS BUFF")
   END_RUNG
   // the same network as SCL:
   IF ("MODE SELECTION DB"."UF PLC_1 MODE BUFF" = 1) AND ("MODE SELECTION DB"."UF PLC_1 PROCESS BUFF" = 125) AND "INPUT MAPPING DB"."ABV 201 FEED BACK CLOSE" THEN
       "MODE SELECTION DB"."UF PLC_1 PROCESS BUFF" := 130;
   END_IF;
END_REGION

REGION Network 29: 135
   RUNG wire#powerrail
      { S7_Templates := "SrcType := Int" } EQ_Contact(in1 := "MODE SELECTION DB"."UF PLC_1 MODE BUFF", in2 := 1)
      { S7_Templates := "SrcType := Int" } EQ_Contact(in1 := "MODE SELECTION DB"."UF PLC_1 PROCESS BUFF", in2 := 130)
      Move(in := 135, out1 => "MODE SELECTION DB"."UF PLC_1 PROCESS BUFF")
   END_RUNG
   // the same network as SCL:
   IF ("MODE SELECTION DB"."UF PLC_1 MODE BUFF" = 1) AND ("MODE SELECTION DB"."UF PLC_1 PROCESS BUFF" = 130) THEN
       "MODE SELECTION DB"."UF PLC_1 PROCESS BUFF" := 135;
   END_IF;
END_REGION

REGION Network 31: ABFV 202 OPEN FB
   RUNG wire#powerrail
      { S7_Templates := "SrcType := Int" } EQ_Contact(in1 := "MODE SELECTION DB"."UF PLC_1 MODE BUFF", in2 := 1)
      { S7_Templates := "SrcType := Int" } EQ_Contact(in1 := "MODE SELECTION DB"."UF PLC_1 PROCESS BUFF", in2 := 135)
      Contact( "INPUT MAPPING DB"."ABFV 202 FEED BACK OPEN" )
      Move(in := 140, out1 => "MODE SELECTION DB"."UF PLC_1 PROCESS BUFF")
   END_RUNG
   // the same network as SCL:
   IF ("MODE SELECTION DB"."UF PLC_1 MODE BUFF" = 1) AND ("MODE SELECTION DB"."UF PLC_1 PROCESS BUFF" = 135) AND "INPUT MAPPING DB"."ABFV 202 FEED BACK OPEN" THEN
       "MODE SELECTION DB"."UF PLC_1 PROCESS BUFF" := 140;
   END_IF;
END_REGION

REGION Network 32: ABFV 203 OPEN FB
   RUNG wire#powerrail
      { S7_Templates := "SrcType := Int" } EQ_Contact(in1 := "MODE SELECTION DB"."UF PLC_1 MODE BUFF", in2 := 1)
      { S7_Templates := "SrcType := Int" } EQ_Contact(in1 := "MODE SELECTION DB"."UF PLC_1 PROCESS BUFF", in2 := 140)
      Contact( "INPUT MAPPING DB"."ABFV 203 FEED BACK OPEN" )
      Move(in := 145, out1 => "MODE SELECTION DB"."UF PLC_1 PROCESS BUFF")
   END_RUNG
   // the same network as SCL:
   IF ("MODE SELECTION DB"."UF PLC_1 MODE BUFF" = 1) AND ("MODE SELECTION DB"."UF PLC_1 PROCESS BUFF" = 140) AND "INPUT MAPPING DB"."ABFV 203 FEED BACK OPEN" THEN
       "MODE SELECTION DB"."UF PLC_1 PROCESS BUFF" := 145;
   END_IF;
END_REGION

REGION Network 33: ABFV 207 OPEN FB
   RUNG wire#powerrail
      { S7_Templates := "SrcType := Int" } EQ_Contact(in1 := "MODE SELECTION DB"."UF PLC_1 MODE BUFF", in2 := 1)
      { S7_Templates := "SrcType := Int" } EQ_Contact(in1 := "MODE SELECTION DB"."UF PLC_1 PROCESS BUFF", in2 := 145)
      Contact( "INPUT MAPPING DB"."ABFV-207 FEED BACK OPEN" )
      { S7_Templates := "time_type := Time" } "IEC_Timer_0_DB_49".TON(pt := T#10S, et =>)
      Move(in := 150, out1 => "MODE SELECTION DB"."UF PLC_1 PROCESS BUFF")
   END_RUNG
   // the same network as SCL:
   "IEC_Timer_0_DB_49".TON(IN := ("MODE SELECTION DB"."UF PLC_1 MODE BUFF" = 1) AND ("MODE SELECTION DB"."UF PLC_1 PROCESS BUFF" = 145) AND "INPUT MAPPING DB"."ABFV-207 FEED BACK OPEN",
                           PT := T#10S);
   IF "IEC_Timer_0_DB_49".Q THEN "MODE SELECTION DB"."UF PLC_1 PROCESS BUFF" := 150; END_IF;
END_REGION

REGION Network 34: DAIN
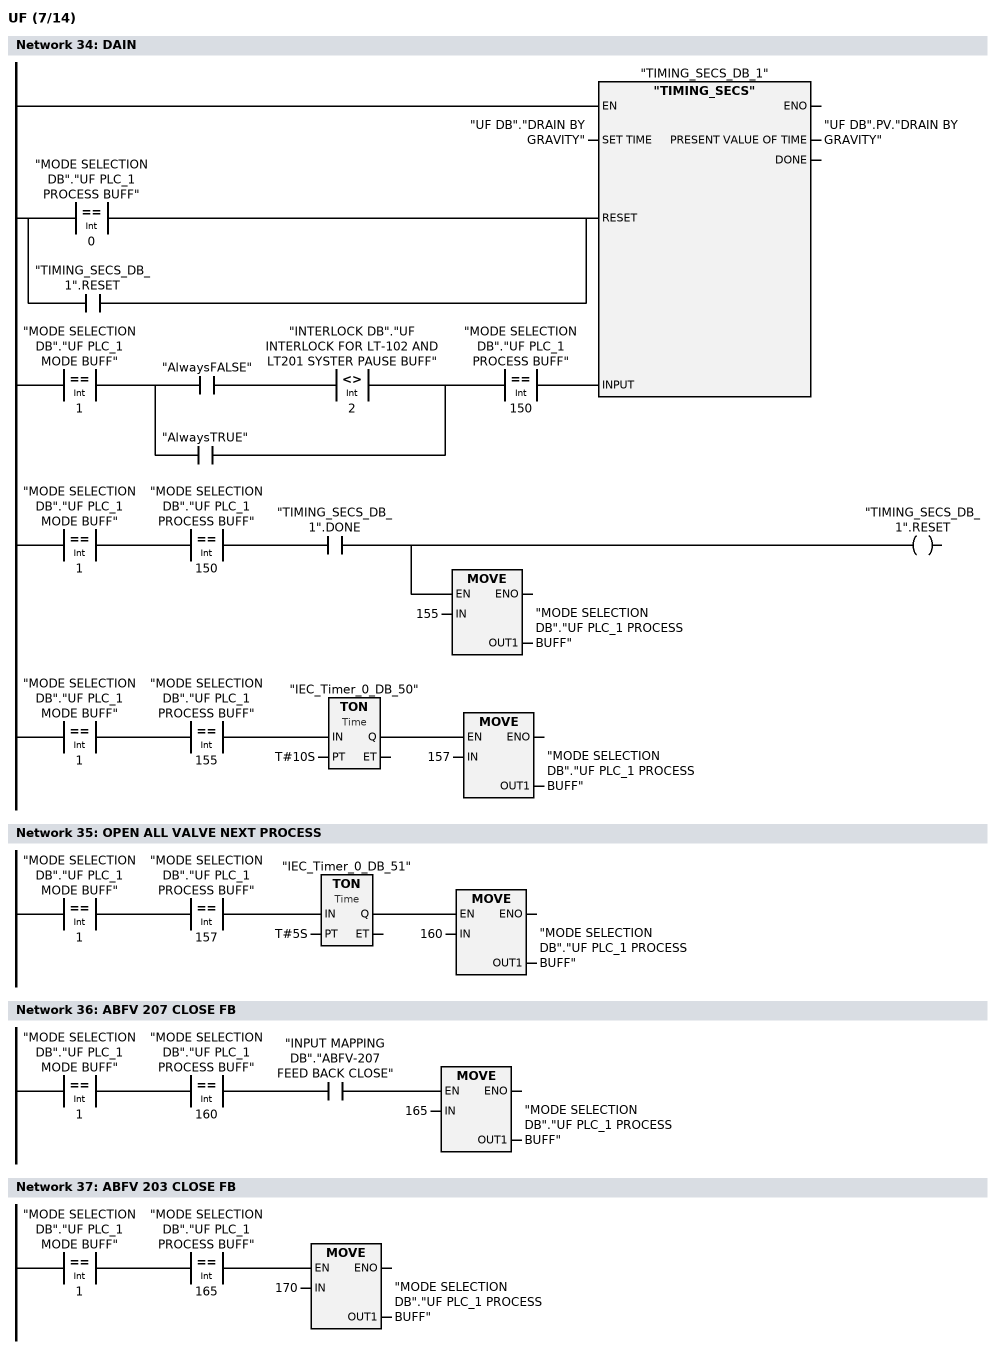
   RUNG wire#powerrail
      "TIMING_SECS_DB_1"(RESET := wire#w1, INPUT := wire#w4, "SET TIME" := "UF DB"."DRAIN BY GRAVITY", "PRESENT VALUE OF TIME" => "UF DB".PV."DRAIN BY GRAVITY", DONE =>)
   END_RUNG
   RUNG wire#powerrail
      { S7_Templates := "SrcType := Int" } EQ_Contact(in1 := "MODE SELECTION DB"."UF PLC_1 PROCESS BUFF", in2 := 0)
   END_RUNG wire#w1
   RUNG wire#powerrail
      Contact( "TIMING_SECS_DB_1".RESET )
   END_RUNG wire#w1
   RUNG wire#powerrail
      { S7_Templates := "SrcType := Int" } EQ_Contact(in1 := "MODE SELECTION DB"."UF PLC_1 MODE BUFF", in2 := 1)
      wire#w2
      Contact( "AlwaysFALSE" )
      { S7_Templates := "SrcType := Int" } NE_Contact(in1 := "INTERLOCK DB"."UF INTERLOCK FOR LT-102 AND LT201 SYSTER PAUSE BUFF", in2 := 2)
      wire#w3
      { S7_Templates := "SrcType := Int" } EQ_Contact(in1 := "MODE SELECTION DB"."UF PLC_1 PROCESS BUFF", in2 := 150)
   END_RUNG wire#w4
   RUNG wire#w2
      Contact( "AlwaysTRUE" )
   END_RUNG wire#w3
   RUNG wire#powerrail
      { S7_Templates := "SrcType := Int" } EQ_Contact(in1 := "MODE SELECTION DB"."UF PLC_1 MODE BUFF", in2 := 1)
      { S7_Templates := "SrcType := Int" } EQ_Contact(in1 := "MODE SELECTION DB"."UF PLC_1 PROCESS BUFF", in2 := 150)
      Contact( "TIMING_SECS_DB_1".DONE )
      wire#w5
      Coil( "TIMING_SECS_DB_1".RESET )
   END_RUNG
   RUNG wire#w5
      Move(in := 155, out1 => "MODE SELECTION DB"."UF PLC_1 PROCESS BUFF")
   END_RUNG
   RUNG wire#powerrail
      { S7_Templates := "SrcType := Int" } EQ_Contact(in1 := "MODE SELECTION DB"."UF PLC_1 MODE BUFF", in2 := 1)
      { S7_Templates := "SrcType := Int" } EQ_Contact(in1 := "MODE SELECTION DB"."UF PLC_1 PROCESS BUFF", in2 := 155)
      { S7_Templates := "time_type := Time" } "IEC_Timer_0_DB_50".TON(pt := T#10S, et =>)
      Move(in := 157, out1 => "MODE SELECTION DB"."UF PLC_1 PROCESS BUFF")
   END_RUNG
   // the same network as SCL:
   "TIMING_SECS_DB_1"("SET TIME" := "UF DB"."DRAIN BY GRAVITY",   // "TIMING_SECS"
                      RESET := ("MODE SELECTION DB"."UF PLC_1 PROCESS BUFF" = 0) OR "TIMING_SECS_DB_1".RESET,
                      INPUT := ("MODE SELECTION DB"."UF PLC_1 MODE BUFF" = 1) AND (("AlwaysFALSE" AND ("INTERLOCK DB"."UF INTERLOCK FOR LT-102 AND LT201 SYSTER PAUSE BUFF" <> 2)) OR "AlwaysTRUE") AND ("MODE SELECTION DB"."UF PLC_1 PROCESS BUFF" = 150),
                      "PRESENT VALUE OF TIME" => "UF DB".PV."DRAIN BY GRAVITY");
   "TIMING_SECS_DB_1".RESET := ("MODE SELECTION DB"."UF PLC_1 MODE BUFF" = 1) AND ("MODE SELECTION DB"."UF PLC_1 PROCESS BUFF" = 150) AND "TIMING_SECS_DB_1".DONE;
   IF "TIMING_SECS_DB_1".RESET THEN "MODE SELECTION DB"."UF PLC_1 PROCESS BUFF" := 155; END_IF;
   "IEC_Timer_0_DB_50".TON(IN := ("MODE SELECTION DB"."UF PLC_1 MODE BUFF" = 1) AND ("MODE SELECTION DB"."UF PLC_1 PROCESS BUFF" = 155),
                           PT := T#10S);
   IF "IEC_Timer_0_DB_50".Q THEN "MODE SELECTION DB"."UF PLC_1 PROCESS BUFF" := 157; END_IF;
END_REGION

REGION Network 35: OPEN ALL VALVE NEXT PROCESS
   RUNG wire#powerrail
      { S7_Templates := "SrcType := Int" } EQ_Contact(in1 := "MODE SELECTION DB"."UF PLC_1 MODE BUFF", in2 := 1)
      { S7_Templates := "SrcType := Int" } EQ_Contact(in1 := "MODE SELECTION DB"."UF PLC_1 PROCESS BUFF", in2 := 157)
      { S7_Templates := "time_type := Time" } "IEC_Timer_0_DB_51".TON(pt := T#5S, et =>)
      Move(in := 160, out1 => "MODE SELECTION DB"."UF PLC_1 PROCESS BUFF")
   END_RUNG
   // the same network as SCL:
   "IEC_Timer_0_DB_51".TON(IN := ("MODE SELECTION DB"."UF PLC_1 MODE BUFF" = 1) AND ("MODE SELECTION DB"."UF PLC_1 PROCESS BUFF" = 157),
                           PT := T#5S);
   IF "IEC_Timer_0_DB_51".Q THEN "MODE SELECTION DB"."UF PLC_1 PROCESS BUFF" := 160; END_IF;
END_REGION

REGION Network 36: ABFV 207 CLOSE FB
   RUNG wire#powerrail
      { S7_Templates := "SrcType := Int" } EQ_Contact(in1 := "MODE SELECTION DB"."UF PLC_1 MODE BUFF", in2 := 1)
      { S7_Templates := "SrcType := Int" } EQ_Contact(in1 := "MODE SELECTION DB"."UF PLC_1 PROCESS BUFF", in2 := 160)
      Contact( "INPUT MAPPING DB"."ABFV-207 FEED BACK CLOSE" )
      Move(in := 165, out1 => "MODE SELECTION DB"."UF PLC_1 PROCESS BUFF")
   END_RUNG
   // the same network as SCL:
   IF ("MODE SELECTION DB"."UF PLC_1 MODE BUFF" = 1) AND ("MODE SELECTION DB"."UF PLC_1 PROCESS BUFF" = 160) AND "INPUT MAPPING DB"."ABFV-207 FEED BACK CLOSE" THEN
       "MODE SELECTION DB"."UF PLC_1 PROCESS BUFF" := 165;
   END_IF;
END_REGION

REGION Network 37: ABFV 203 CLOSE FB
   RUNG wire#powerrail
      { S7_Templates := "SrcType := Int" } EQ_Contact(in1 := "MODE SELECTION DB"."UF PLC_1 MODE BUFF", in2 := 1)
      { S7_Templates := "SrcType := Int" } EQ_Contact(in1 := "MODE SELECTION DB"."UF PLC_1 PROCESS BUFF", in2 := 165)
      Move(in := 170, out1 => "MODE SELECTION DB"."UF PLC_1 PROCESS BUFF")
   END_RUNG
   // the same network as SCL:
   IF ("MODE SELECTION DB"."UF PLC_1 MODE BUFF" = 1) AND ("MODE SELECTION DB"."UF PLC_1 PROCESS BUFF" = 165) THEN
       "MODE SELECTION DB"."UF PLC_1 PROCESS BUFF" := 170;
   END_IF;
END_REGION

REGION Network 38: ABFV 202 CLOSE FB
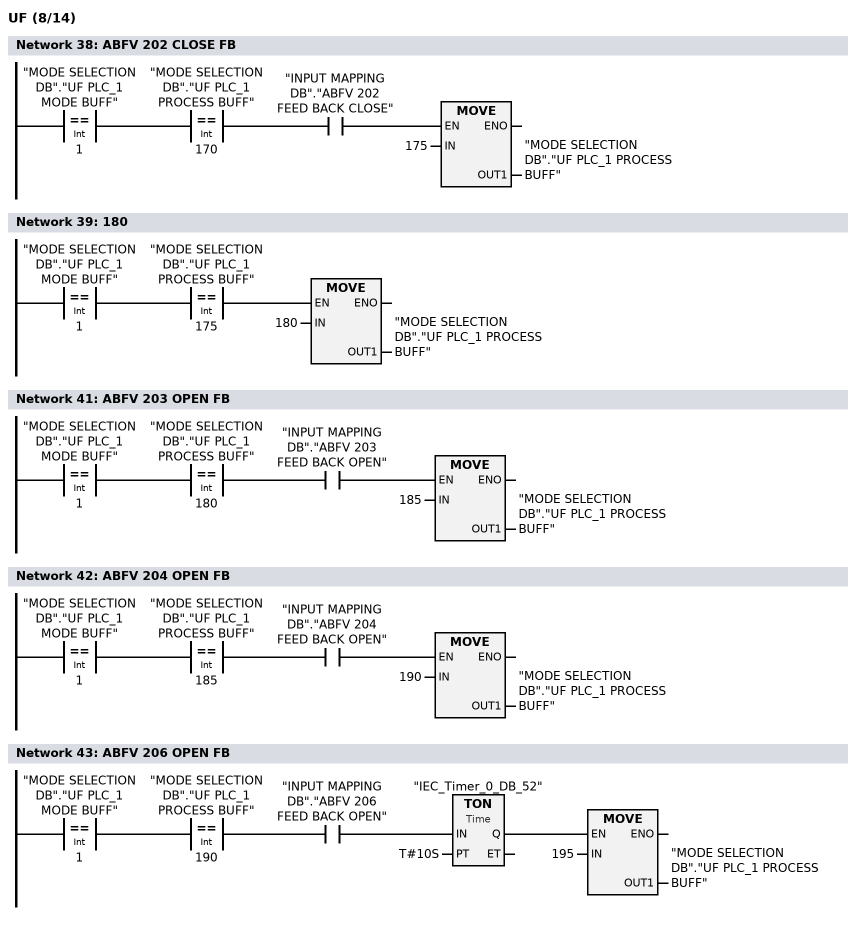
   RUNG wire#powerrail
      { S7_Templates := "SrcType := Int" } EQ_Contact(in1 := "MODE SELECTION DB"."UF PLC_1 MODE BUFF", in2 := 1)
      { S7_Templates := "SrcType := Int" } EQ_Contact(in1 := "MODE SELECTION DB"."UF PLC_1 PROCESS BUFF", in2 := 170)
      Contact( "INPUT MAPPING DB"."ABFV 202 FEED BACK CLOSE" )
      Move(in := 175, out1 => "MODE SELECTION DB"."UF PLC_1 PROCESS BUFF")
   END_RUNG
   // the same network as SCL:
   IF ("MODE SELECTION DB"."UF PLC_1 MODE BUFF" = 1) AND ("MODE SELECTION DB"."UF PLC_1 PROCESS BUFF" = 170) AND "INPUT MAPPING DB"."ABFV 202 FEED BACK CLOSE" THEN
       "MODE SELECTION DB"."UF PLC_1 PROCESS BUFF" := 175;
   END_IF;
END_REGION

REGION Network 39: 180
   RUNG wire#powerrail
      { S7_Templates := "SrcType := Int" } EQ_Contact(in1 := "MODE SELECTION DB"."UF PLC_1 MODE BUFF", in2 := 1)
      { S7_Templates := "SrcType := Int" } EQ_Contact(in1 := "MODE SELECTION DB"."UF PLC_1 PROCESS BUFF", in2 := 175)
      Move(in := 180, out1 => "MODE SELECTION DB"."UF PLC_1 PROCESS BUFF")
   END_RUNG
   // the same network as SCL:
   IF ("MODE SELECTION DB"."UF PLC_1 MODE BUFF" = 1) AND ("MODE SELECTION DB"."UF PLC_1 PROCESS BUFF" = 175) THEN
       "MODE SELECTION DB"."UF PLC_1 PROCESS BUFF" := 180;
   END_IF;
END_REGION

REGION Network 41: ABFV 203 OPEN FB
   RUNG wire#powerrail
      { S7_Templates := "SrcType := Int" } EQ_Contact(in1 := "MODE SELECTION DB"."UF PLC_1 MODE BUFF", in2 := 1)
      { S7_Templates := "SrcType := Int" } EQ_Contact(in1 := "MODE SELECTION DB"."UF PLC_1 PROCESS BUFF", in2 := 180)
      Contact( "INPUT MAPPING DB"."ABFV 203 FEED BACK OPEN" )
      Move(in := 185, out1 => "MODE SELECTION DB"."UF PLC_1 PROCESS BUFF")
   END_RUNG
   // the same network as SCL:
   IF ("MODE SELECTION DB"."UF PLC_1 MODE BUFF" = 1) AND ("MODE SELECTION DB"."UF PLC_1 PROCESS BUFF" = 180) AND "INPUT MAPPING DB"."ABFV 203 FEED BACK OPEN" THEN
       "MODE SELECTION DB"."UF PLC_1 PROCESS BUFF" := 185;
   END_IF;
END_REGION

REGION Network 42: ABFV 204 OPEN FB
   RUNG wire#powerrail
      { S7_Templates := "SrcType := Int" } EQ_Contact(in1 := "MODE SELECTION DB"."UF PLC_1 MODE BUFF", in2 := 1)
      { S7_Templates := "SrcType := Int" } EQ_Contact(in1 := "MODE SELECTION DB"."UF PLC_1 PROCESS BUFF", in2 := 185)
      Contact( "INPUT MAPPING DB"."ABFV 204 FEED BACK OPEN" )
      Move(in := 190, out1 => "MODE SELECTION DB"."UF PLC_1 PROCESS BUFF")
   END_RUNG
   // the same network as SCL:
   IF ("MODE SELECTION DB"."UF PLC_1 MODE BUFF" = 1) AND ("MODE SELECTION DB"."UF PLC_1 PROCESS BUFF" = 185) AND "INPUT MAPPING DB"."ABFV 204 FEED BACK OPEN" THEN
       "MODE SELECTION DB"."UF PLC_1 PROCESS BUFF" := 190;
   END_IF;
END_REGION

REGION Network 43: ABFV 206 OPEN FB
   RUNG wire#powerrail
      { S7_Templates := "SrcType := Int" } EQ_Contact(in1 := "MODE SELECTION DB"."UF PLC_1 MODE BUFF", in2 := 1)
      { S7_Templates := "SrcType := Int" } EQ_Contact(in1 := "MODE SELECTION DB"."UF PLC_1 PROCESS BUFF", in2 := 190)
      Contact( "INPUT MAPPING DB"."ABFV 206 FEED BACK OPEN" )
      { S7_Templates := "time_type := Time" } "IEC_Timer_0_DB_52".TON(pt := T#10S, et =>)
      Move(in := 195, out1 => "MODE SELECTION DB"."UF PLC_1 PROCESS BUFF")
   END_RUNG
   // the same network as SCL:
   "IEC_Timer_0_DB_52".TON(IN := ("MODE SELECTION DB"."UF PLC_1 MODE BUFF" = 1) AND ("MODE SELECTION DB"."UF PLC_1 PROCESS BUFF" = 190) AND "INPUT MAPPING DB"."ABFV 206 FEED BACK OPEN",
                           PT := T#10S);
   IF "IEC_Timer_0_DB_52".Q THEN "MODE SELECTION DB"."UF PLC_1 PROCESS BUFF" := 195; END_IF;
END_REGION

REGION Network 44: BACKWASH-1
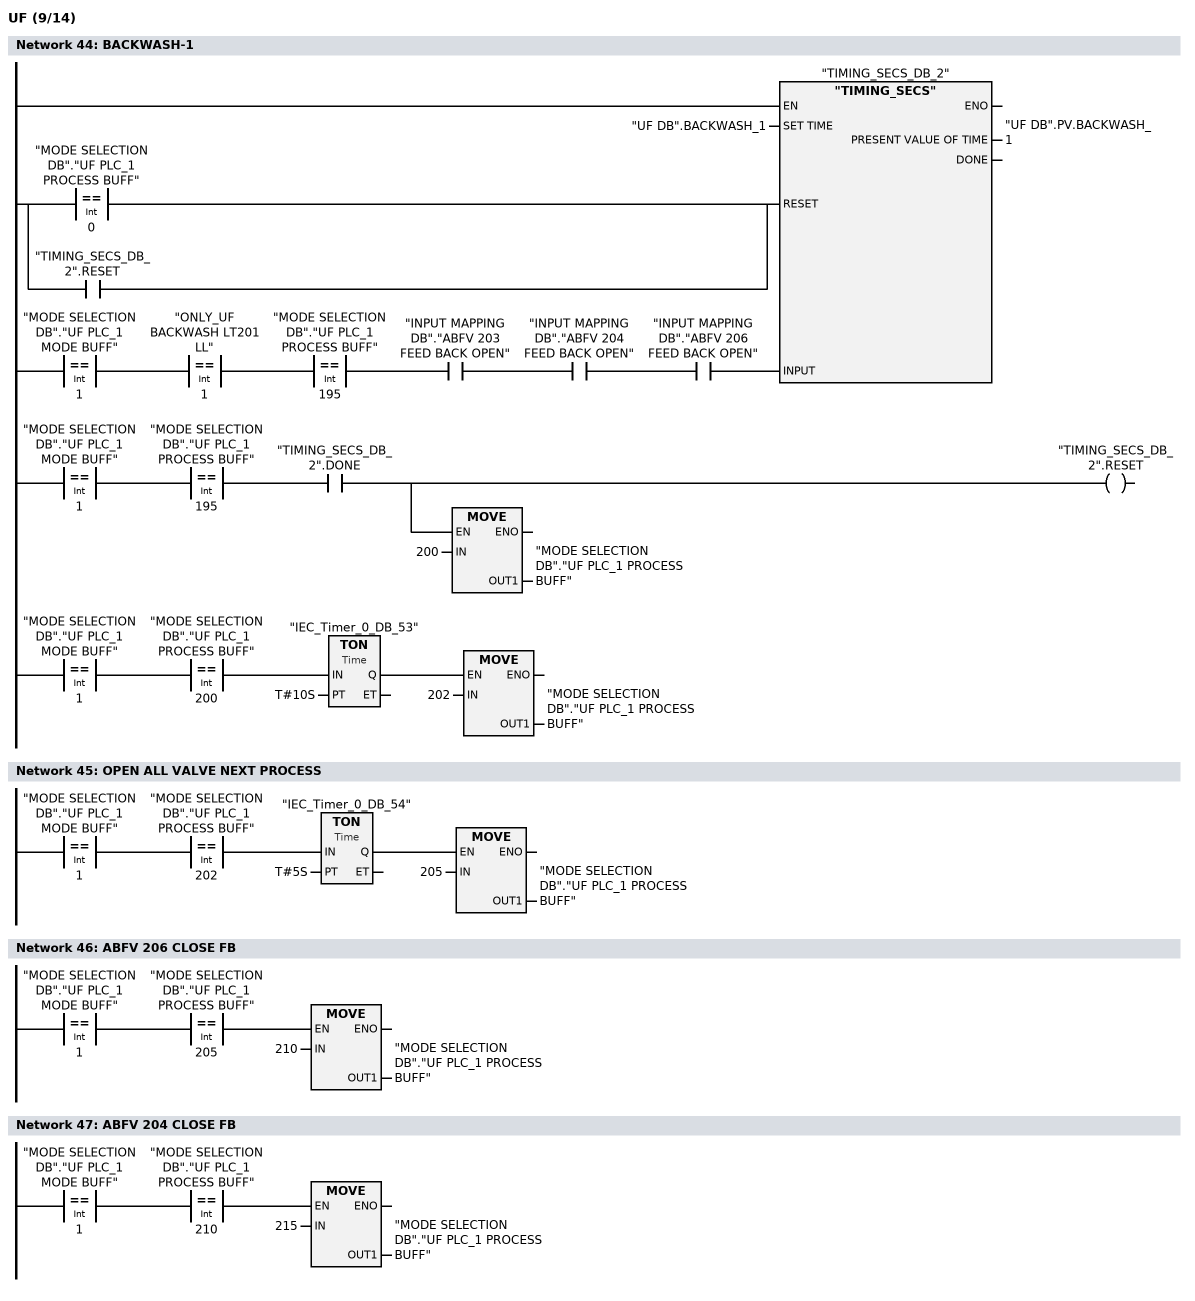
   RUNG wire#powerrail
      "TIMING_SECS_DB_2"(RESET := wire#w1, INPUT := wire#w2, "SET TIME" := "UF DB".BACKWASH_1, "PRESENT VALUE OF TIME" => "UF DB".PV.BACKWASH_1, DONE =>)
   END_RUNG
   RUNG wire#powerrail
      { S7_Templates := "SrcType := Int" } EQ_Contact(in1 := "MODE SELECTION DB"."UF PLC_1 PROCESS BUFF", in2 := 0)
   END_RUNG wire#w1
   RUNG wire#powerrail
      Contact( "TIMING_SECS_DB_2".RESET )
   END_RUNG wire#w1
   RUNG wire#powerrail
      { S7_Templates := "SrcType := Int" } EQ_Contact(in1 := "MODE SELECTION DB"."UF PLC_1 MODE BUFF", in2 := 1)
      { S7_Templates := "SrcType := Int" } EQ_Contact(in1 := "ONLY_UF BACKWASH LT201 LL", in2 := 1)
      { S7_Templates := "SrcType := Int" } EQ_Contact(in1 := "MODE SELECTION DB"."UF PLC_1 PROCESS BUFF", in2 := 195)
      Contact( "INPUT MAPPING DB"."ABFV 203 FEED BACK OPEN" )
      Contact( "INPUT MAPPING DB"."ABFV 204 FEED BACK OPEN" )
      Contact( "INPUT MAPPING DB"."ABFV 206 FEED BACK OPEN" )
   END_RUNG wire#w2
   RUNG wire#powerrail
      { S7_Templates := "SrcType := Int" } EQ_Contact(in1 := "MODE SELECTION DB"."UF PLC_1 MODE BUFF", in2 := 1)
      { S7_Templates := "SrcType := Int" } EQ_Contact(in1 := "MODE SELECTION DB"."UF PLC_1 PROCESS BUFF", in2 := 195)
      Contact( "TIMING_SECS_DB_2".DONE )
      wire#w3
      Coil( "TIMING_SECS_DB_2".RESET )
   END_RUNG
   RUNG wire#w3
      Move(in := 200, out1 => "MODE SELECTION DB"."UF PLC_1 PROCESS BUFF")
   END_RUNG
   RUNG wire#powerrail
      { S7_Templates := "SrcType := Int" } EQ_Contact(in1 := "MODE SELECTION DB"."UF PLC_1 MODE BUFF", in2 := 1)
      { S7_Templates := "SrcType := Int" } EQ_Contact(in1 := "MODE SELECTION DB"."UF PLC_1 PROCESS BUFF", in2 := 200)
      { S7_Templates := "time_type := Time" } "IEC_Timer_0_DB_53".TON(pt := T#10S, et =>)
      Move(in := 202, out1 => "MODE SELECTION DB"."UF PLC_1 PROCESS BUFF")
   END_RUNG
   // the same network as SCL:
   "TIMING_SECS_DB_2"("SET TIME" := "UF DB".BACKWASH_1,   // "TIMING_SECS"
                      RESET := ("MODE SELECTION DB"."UF PLC_1 PROCESS BUFF" = 0) OR "TIMING_SECS_DB_2".RESET,
                      INPUT := ("MODE SELECTION DB"."UF PLC_1 MODE BUFF" = 1) AND ("ONLY_UF BACKWASH LT201 LL" = 1) AND ("MODE SELECTION DB"."UF PLC_1 PROCESS BUFF" = 195) AND "INPUT MAPPING DB"."ABFV 203 FEED BACK OPEN" AND "INPUT MAPPING DB"."ABFV 204 FEED BACK OPEN" AND "INPUT MAPPING DB"."ABFV 206 FEED BACK OPEN",
                      "PRESENT VALUE OF TIME" => "UF DB".PV.BACKWASH_1);
   "TIMING_SECS_DB_2".RESET := ("MODE SELECTION DB"."UF PLC_1 MODE BUFF" = 1) AND ("MODE SELECTION DB"."UF PLC_1 PROCESS BUFF" = 195) AND "TIMING_SECS_DB_2".DONE;
   IF "TIMING_SECS_DB_2".RESET THEN "MODE SELECTION DB"."UF PLC_1 PROCESS BUFF" := 200; END_IF;
   "IEC_Timer_0_DB_53".TON(IN := ("MODE SELECTION DB"."UF PLC_1 MODE BUFF" = 1) AND ("MODE SELECTION DB"."UF PLC_1 PROCESS BUFF" = 200),
                           PT := T#10S);
   IF "IEC_Timer_0_DB_53".Q THEN "MODE SELECTION DB"."UF PLC_1 PROCESS BUFF" := 202; END_IF;
END_REGION

REGION Network 45: OPEN ALL VALVE NEXT PROCESS
   RUNG wire#powerrail
      { S7_Templates := "SrcType := Int" } EQ_Contact(in1 := "MODE SELECTION DB"."UF PLC_1 MODE BUFF", in2 := 1)
      { S7_Templates := "SrcType := Int" } EQ_Contact(in1 := "MODE SELECTION DB"."UF PLC_1 PROCESS BUFF", in2 := 202)
      { S7_Templates := "time_type := Time" } "IEC_Timer_0_DB_54".TON(pt := T#5S, et =>)
      Move(in := 205, out1 => "MODE SELECTION DB"."UF PLC_1 PROCESS BUFF")
   END_RUNG
   // the same network as SCL:
   "IEC_Timer_0_DB_54".TON(IN := ("MODE SELECTION DB"."UF PLC_1 MODE BUFF" = 1) AND ("MODE SELECTION DB"."UF PLC_1 PROCESS BUFF" = 202),
                           PT := T#5S);
   IF "IEC_Timer_0_DB_54".Q THEN "MODE SELECTION DB"."UF PLC_1 PROCESS BUFF" := 205; END_IF;
END_REGION

REGION Network 46: ABFV 206 CLOSE FB
   RUNG wire#powerrail
      { S7_Templates := "SrcType := Int" } EQ_Contact(in1 := "MODE SELECTION DB"."UF PLC_1 MODE BUFF", in2 := 1)
      { S7_Templates := "SrcType := Int" } EQ_Contact(in1 := "MODE SELECTION DB"."UF PLC_1 PROCESS BUFF", in2 := 205)
      Move(in := 210, out1 => "MODE SELECTION DB"."UF PLC_1 PROCESS BUFF")
   END_RUNG
   // the same network as SCL:
   IF ("MODE SELECTION DB"."UF PLC_1 MODE BUFF" = 1) AND ("MODE SELECTION DB"."UF PLC_1 PROCESS BUFF" = 205) THEN
       "MODE SELECTION DB"."UF PLC_1 PROCESS BUFF" := 210;
   END_IF;
END_REGION

REGION Network 47: ABFV 204 CLOSE FB
   RUNG wire#powerrail
      { S7_Templates := "SrcType := Int" } EQ_Contact(in1 := "MODE SELECTION DB"."UF PLC_1 MODE BUFF", in2 := 1)
      { S7_Templates := "SrcType := Int" } EQ_Contact(in1 := "MODE SELECTION DB"."UF PLC_1 PROCESS BUFF", in2 := 210)
      Move(in := 215, out1 => "MODE SELECTION DB"."UF PLC_1 PROCESS BUFF")
   END_RUNG
   // the same network as SCL:
   IF ("MODE SELECTION DB"."UF PLC_1 MODE BUFF" = 1) AND ("MODE SELECTION DB"."UF PLC_1 PROCESS BUFF" = 210) THEN
       "MODE SELECTION DB"."UF PLC_1 PROCESS BUFF" := 215;
   END_IF;
END_REGION

REGION Network 48: ABFV 203 CLOSE FB
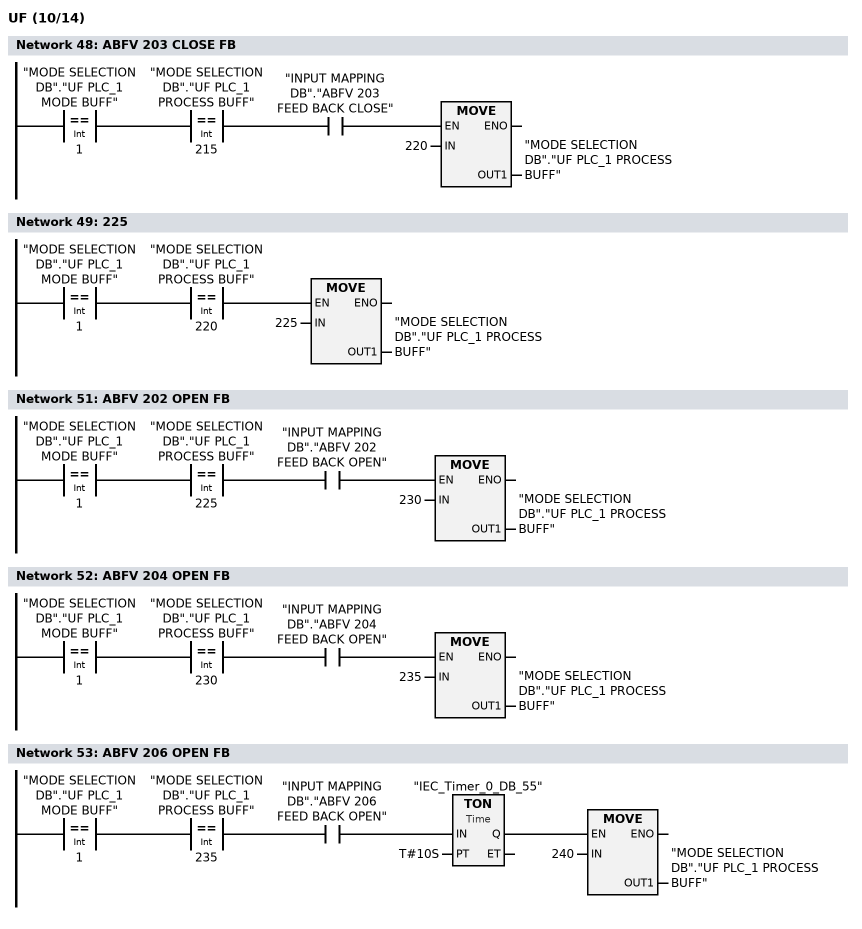
   RUNG wire#powerrail
      { S7_Templates := "SrcType := Int" } EQ_Contact(in1 := "MODE SELECTION DB"."UF PLC_1 MODE BUFF", in2 := 1)
      { S7_Templates := "SrcType := Int" } EQ_Contact(in1 := "MODE SELECTION DB"."UF PLC_1 PROCESS BUFF", in2 := 215)
      Contact( "INPUT MAPPING DB"."ABFV 203 FEED BACK CLOSE" )
      Move(in := 220, out1 => "MODE SELECTION DB"."UF PLC_1 PROCESS BUFF")
   END_RUNG
   // the same network as SCL:
   IF ("MODE SELECTION DB"."UF PLC_1 MODE BUFF" = 1) AND ("MODE SELECTION DB"."UF PLC_1 PROCESS BUFF" = 215) AND "INPUT MAPPING DB"."ABFV 203 FEED BACK CLOSE" THEN
       "MODE SELECTION DB"."UF PLC_1 PROCESS BUFF" := 220;
   END_IF;
END_REGION

REGION Network 49: 225
   RUNG wire#powerrail
      { S7_Templates := "SrcType := Int" } EQ_Contact(in1 := "MODE SELECTION DB"."UF PLC_1 MODE BUFF", in2 := 1)
      { S7_Templates := "SrcType := Int" } EQ_Contact(in1 := "MODE SELECTION DB"."UF PLC_1 PROCESS BUFF", in2 := 220)
      Move(in := 225, out1 => "MODE SELECTION DB"."UF PLC_1 PROCESS BUFF")
   END_RUNG
   // the same network as SCL:
   IF ("MODE SELECTION DB"."UF PLC_1 MODE BUFF" = 1) AND ("MODE SELECTION DB"."UF PLC_1 PROCESS BUFF" = 220) THEN
       "MODE SELECTION DB"."UF PLC_1 PROCESS BUFF" := 225;
   END_IF;
END_REGION

REGION Network 51: ABFV 202 OPEN FB
   RUNG wire#powerrail
      { S7_Templates := "SrcType := Int" } EQ_Contact(in1 := "MODE SELECTION DB"."UF PLC_1 MODE BUFF", in2 := 1)
      { S7_Templates := "SrcType := Int" } EQ_Contact(in1 := "MODE SELECTION DB"."UF PLC_1 PROCESS BUFF", in2 := 225)
      Contact( "INPUT MAPPING DB"."ABFV 202 FEED BACK OPEN" )
      Move(in := 230, out1 => "MODE SELECTION DB"."UF PLC_1 PROCESS BUFF")
   END_RUNG
   // the same network as SCL:
   IF ("MODE SELECTION DB"."UF PLC_1 MODE BUFF" = 1) AND ("MODE SELECTION DB"."UF PLC_1 PROCESS BUFF" = 225) AND "INPUT MAPPING DB"."ABFV 202 FEED BACK OPEN" THEN
       "MODE SELECTION DB"."UF PLC_1 PROCESS BUFF" := 230;
   END_IF;
END_REGION

REGION Network 52: ABFV 204 OPEN FB
   RUNG wire#powerrail
      { S7_Templates := "SrcType := Int" } EQ_Contact(in1 := "MODE SELECTION DB"."UF PLC_1 MODE BUFF", in2 := 1)
      { S7_Templates := "SrcType := Int" } EQ_Contact(in1 := "MODE SELECTION DB"."UF PLC_1 PROCESS BUFF", in2 := 230)
      Contact( "INPUT MAPPING DB"."ABFV 204 FEED BACK OPEN" )
      Move(in := 235, out1 => "MODE SELECTION DB"."UF PLC_1 PROCESS BUFF")
   END_RUNG
   // the same network as SCL:
   IF ("MODE SELECTION DB"."UF PLC_1 MODE BUFF" = 1) AND ("MODE SELECTION DB"."UF PLC_1 PROCESS BUFF" = 230) AND "INPUT MAPPING DB"."ABFV 204 FEED BACK OPEN" THEN
       "MODE SELECTION DB"."UF PLC_1 PROCESS BUFF" := 235;
   END_IF;
END_REGION

REGION Network 53: ABFV 206 OPEN FB
   RUNG wire#powerrail
      { S7_Templates := "SrcType := Int" } EQ_Contact(in1 := "MODE SELECTION DB"."UF PLC_1 MODE BUFF", in2 := 1)
      { S7_Templates := "SrcType := Int" } EQ_Contact(in1 := "MODE SELECTION DB"."UF PLC_1 PROCESS BUFF", in2 := 235)
      Contact( "INPUT MAPPING DB"."ABFV 206 FEED BACK OPEN" )
      { S7_Templates := "time_type := Time" } "IEC_Timer_0_DB_55".TON(pt := T#10S, et =>)
      Move(in := 240, out1 => "MODE SELECTION DB"."UF PLC_1 PROCESS BUFF")
   END_RUNG
   // the same network as SCL:
   "IEC_Timer_0_DB_55".TON(IN := ("MODE SELECTION DB"."UF PLC_1 MODE BUFF" = 1) AND ("MODE SELECTION DB"."UF PLC_1 PROCESS BUFF" = 235) AND "INPUT MAPPING DB"."ABFV 206 FEED BACK OPEN",
                           PT := T#10S);
   IF "IEC_Timer_0_DB_55".Q THEN "MODE SELECTION DB"."UF PLC_1 PROCESS BUFF" := 240; END_IF;
END_REGION

REGION Network 54: BACKWASH-2
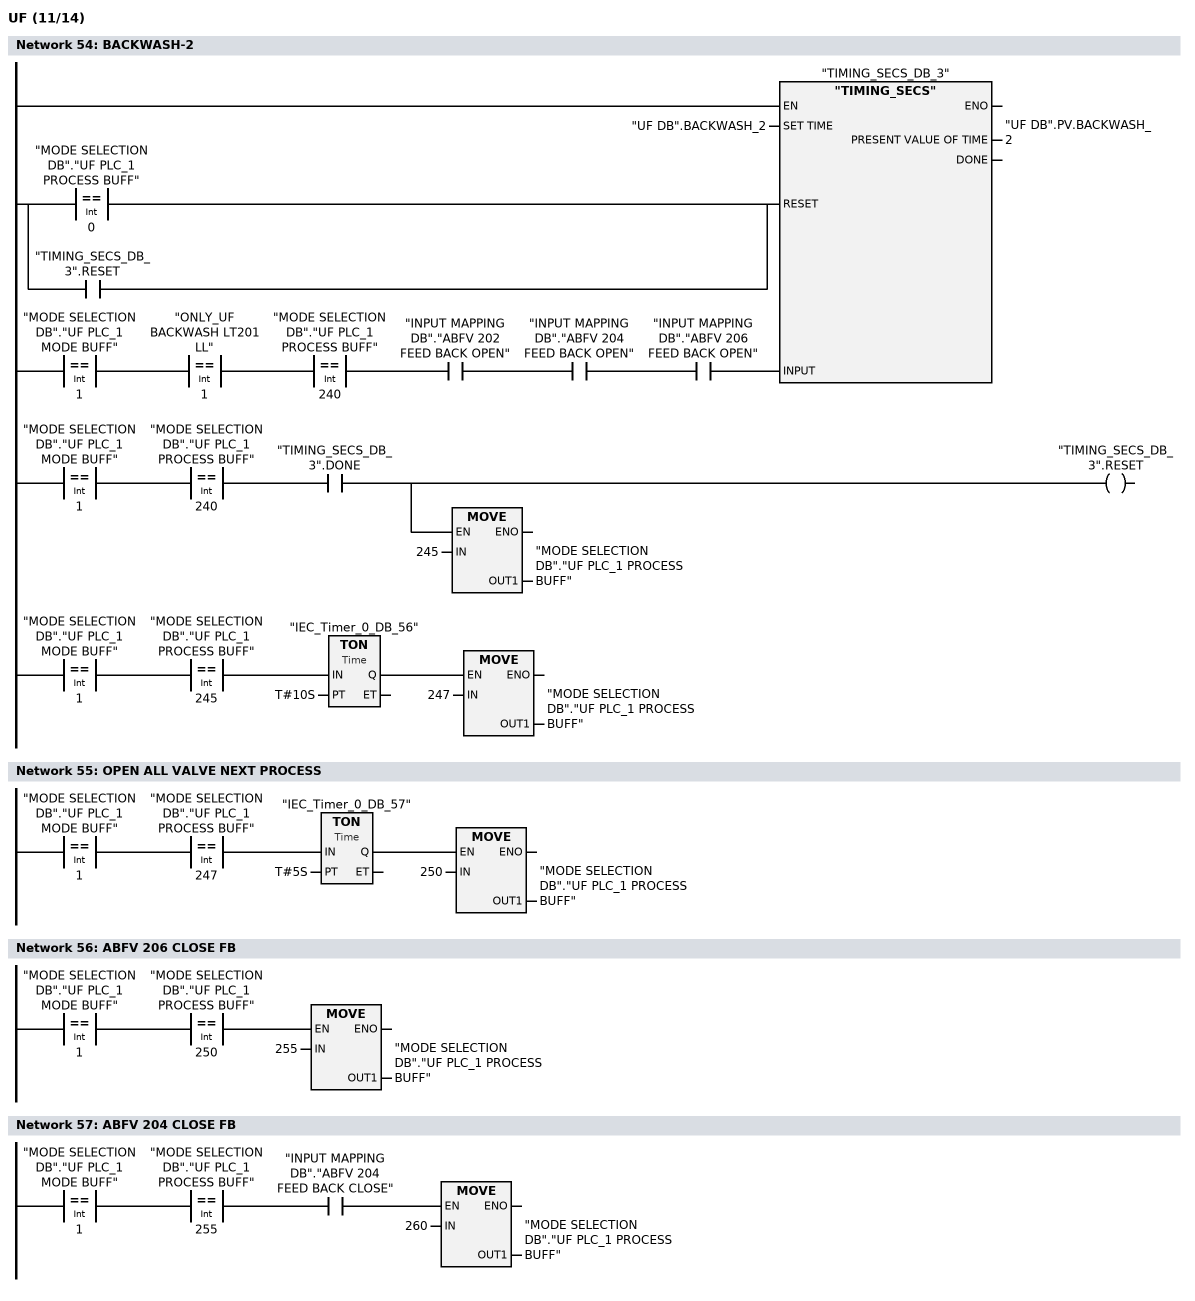
   RUNG wire#powerrail
      "TIMING_SECS_DB_3"(RESET := wire#w1, INPUT := wire#w2, "SET TIME" := "UF DB".BACKWASH_2, "PRESENT VALUE OF TIME" => "UF DB".PV.BACKWASH_2, DONE =>)
   END_RUNG
   RUNG wire#powerrail
      { S7_Templates := "SrcType := Int" } EQ_Contact(in1 := "MODE SELECTION DB"."UF PLC_1 PROCESS BUFF", in2 := 0)
   END_RUNG wire#w1
   RUNG wire#powerrail
      Contact( "TIMING_SECS_DB_3".RESET )
   END_RUNG wire#w1
   RUNG wire#powerrail
      { S7_Templates := "SrcType := Int" } EQ_Contact(in1 := "MODE SELECTION DB"."UF PLC_1 MODE BUFF", in2 := 1)
      { S7_Templates := "SrcType := Int" } EQ_Contact(in1 := "ONLY_UF BACKWASH LT201 LL", in2 := 1)
      { S7_Templates := "SrcType := Int" } EQ_Contact(in1 := "MODE SELECTION DB"."UF PLC_1 PROCESS BUFF", in2 := 240)
      Contact( "INPUT MAPPING DB"."ABFV 202 FEED BACK OPEN" )
      Contact( "INPUT MAPPING DB"."ABFV 204 FEED BACK OPEN" )
      Contact( "INPUT MAPPING DB"."ABFV 206 FEED BACK OPEN" )
   END_RUNG wire#w2
   RUNG wire#powerrail
      { S7_Templates := "SrcType := Int" } EQ_Contact(in1 := "MODE SELECTION DB"."UF PLC_1 MODE BUFF", in2 := 1)
      { S7_Templates := "SrcType := Int" } EQ_Contact(in1 := "MODE SELECTION DB"."UF PLC_1 PROCESS BUFF", in2 := 240)
      Contact( "TIMING_SECS_DB_3".DONE )
      wire#w3
      Coil( "TIMING_SECS_DB_3".RESET )
   END_RUNG
   RUNG wire#w3
      Move(in := 245, out1 => "MODE SELECTION DB"."UF PLC_1 PROCESS BUFF")
   END_RUNG
   RUNG wire#powerrail
      { S7_Templates := "SrcType := Int" } EQ_Contact(in1 := "MODE SELECTION DB"."UF PLC_1 MODE BUFF", in2 := 1)
      { S7_Templates := "SrcType := Int" } EQ_Contact(in1 := "MODE SELECTION DB"."UF PLC_1 PROCESS BUFF", in2 := 245)
      { S7_Templates := "time_type := Time" } "IEC_Timer_0_DB_56".TON(pt := T#10S, et =>)
      Move(in := 247, out1 => "MODE SELECTION DB"."UF PLC_1 PROCESS BUFF")
   END_RUNG
   // the same network as SCL:
   "TIMING_SECS_DB_3"("SET TIME" := "UF DB".BACKWASH_2,   // "TIMING_SECS"
                      RESET := ("MODE SELECTION DB"."UF PLC_1 PROCESS BUFF" = 0) OR "TIMING_SECS_DB_3".RESET,
                      INPUT := ("MODE SELECTION DB"."UF PLC_1 MODE BUFF" = 1) AND ("ONLY_UF BACKWASH LT201 LL" = 1) AND ("MODE SELECTION DB"."UF PLC_1 PROCESS BUFF" = 240) AND "INPUT MAPPING DB"."ABFV 202 FEED BACK OPEN" AND "INPUT MAPPING DB"."ABFV 204 FEED BACK OPEN" AND "INPUT MAPPING DB"."ABFV 206 FEED BACK OPEN",
                      "PRESENT VALUE OF TIME" => "UF DB".PV.BACKWASH_2);
   "TIMING_SECS_DB_3".RESET := ("MODE SELECTION DB"."UF PLC_1 MODE BUFF" = 1) AND ("MODE SELECTION DB"."UF PLC_1 PROCESS BUFF" = 240) AND "TIMING_SECS_DB_3".DONE;
   IF "TIMING_SECS_DB_3".RESET THEN "MODE SELECTION DB"."UF PLC_1 PROCESS BUFF" := 245; END_IF;
   "IEC_Timer_0_DB_56".TON(IN := ("MODE SELECTION DB"."UF PLC_1 MODE BUFF" = 1) AND ("MODE SELECTION DB"."UF PLC_1 PROCESS BUFF" = 245),
                           PT := T#10S);
   IF "IEC_Timer_0_DB_56".Q THEN "MODE SELECTION DB"."UF PLC_1 PROCESS BUFF" := 247; END_IF;
END_REGION

REGION Network 55: OPEN ALL VALVE NEXT PROCESS
   RUNG wire#powerrail
      { S7_Templates := "SrcType := Int" } EQ_Contact(in1 := "MODE SELECTION DB"."UF PLC_1 MODE BUFF", in2 := 1)
      { S7_Templates := "SrcType := Int" } EQ_Contact(in1 := "MODE SELECTION DB"."UF PLC_1 PROCESS BUFF", in2 := 247)
      { S7_Templates := "time_type := Time" } "IEC_Timer_0_DB_57".TON(pt := T#5S, et =>)
      Move(in := 250, out1 => "MODE SELECTION DB"."UF PLC_1 PROCESS BUFF")
   END_RUNG
   // the same network as SCL:
   "IEC_Timer_0_DB_57".TON(IN := ("MODE SELECTION DB"."UF PLC_1 MODE BUFF" = 1) AND ("MODE SELECTION DB"."UF PLC_1 PROCESS BUFF" = 247),
                           PT := T#5S);
   IF "IEC_Timer_0_DB_57".Q THEN "MODE SELECTION DB"."UF PLC_1 PROCESS BUFF" := 250; END_IF;
END_REGION

REGION Network 56: ABFV 206 CLOSE FB
   RUNG wire#powerrail
      { S7_Templates := "SrcType := Int" } EQ_Contact(in1 := "MODE SELECTION DB"."UF PLC_1 MODE BUFF", in2 := 1)
      { S7_Templates := "SrcType := Int" } EQ_Contact(in1 := "MODE SELECTION DB"."UF PLC_1 PROCESS BUFF", in2 := 250)
      Move(in := 255, out1 => "MODE SELECTION DB"."UF PLC_1 PROCESS BUFF")
   END_RUNG
   // the same network as SCL:
   IF ("MODE SELECTION DB"."UF PLC_1 MODE BUFF" = 1) AND ("MODE SELECTION DB"."UF PLC_1 PROCESS BUFF" = 250) THEN
       "MODE SELECTION DB"."UF PLC_1 PROCESS BUFF" := 255;
   END_IF;
END_REGION

REGION Network 57: ABFV 204 CLOSE FB
   RUNG wire#powerrail
      { S7_Templates := "SrcType := Int" } EQ_Contact(in1 := "MODE SELECTION DB"."UF PLC_1 MODE BUFF", in2 := 1)
      { S7_Templates := "SrcType := Int" } EQ_Contact(in1 := "MODE SELECTION DB"."UF PLC_1 PROCESS BUFF", in2 := 255)
      Contact( "INPUT MAPPING DB"."ABFV 204 FEED BACK CLOSE" )
      Move(in := 260, out1 => "MODE SELECTION DB"."UF PLC_1 PROCESS BUFF")
   END_RUNG
   // the same network as SCL:
   IF ("MODE SELECTION DB"."UF PLC_1 MODE BUFF" = 1) AND ("MODE SELECTION DB"."UF PLC_1 PROCESS BUFF" = 255) AND "INPUT MAPPING DB"."ABFV 204 FEED BACK CLOSE" THEN
       "MODE SELECTION DB"."UF PLC_1 PROCESS BUFF" := 260;
   END_IF;
END_REGION

REGION Network 58: ABFV 202 CLOSE FB
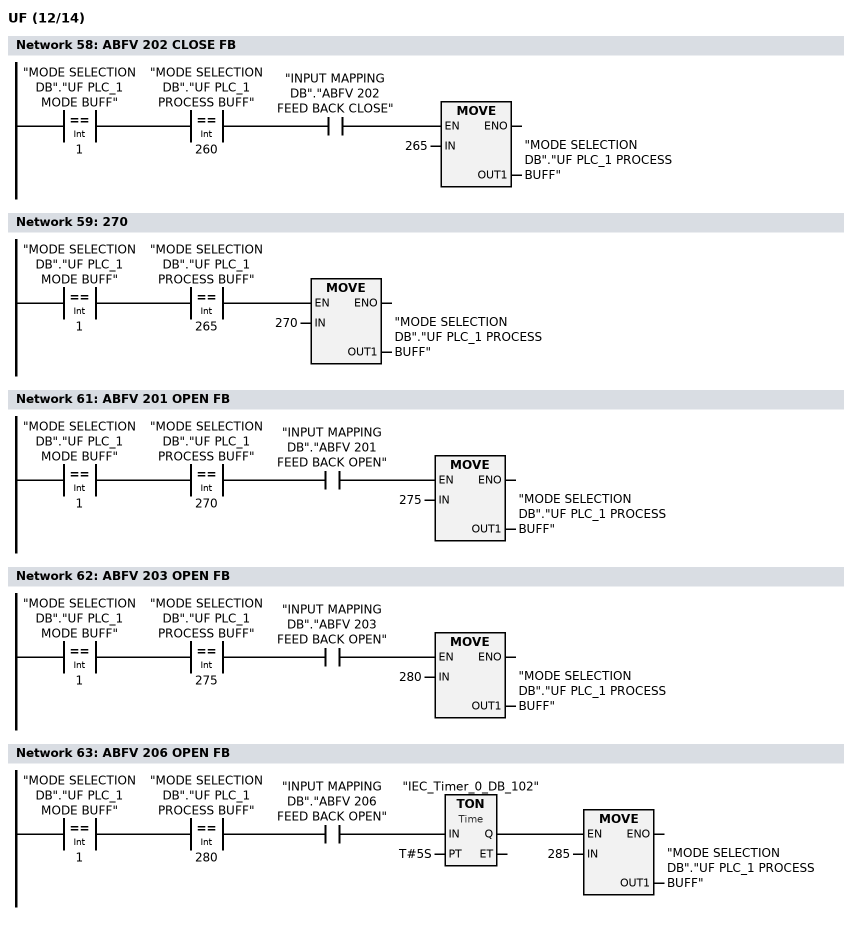
   RUNG wire#powerrail
      { S7_Templates := "SrcType := Int" } EQ_Contact(in1 := "MODE SELECTION DB"."UF PLC_1 MODE BUFF", in2 := 1)
      { S7_Templates := "SrcType := Int" } EQ_Contact(in1 := "MODE SELECTION DB"."UF PLC_1 PROCESS BUFF", in2 := 260)
      Contact( "INPUT MAPPING DB"."ABFV 202 FEED BACK CLOSE" )
      Move(in := 265, out1 => "MODE SELECTION DB"."UF PLC_1 PROCESS BUFF")
   END_RUNG
   // the same network as SCL:
   IF ("MODE SELECTION DB"."UF PLC_1 MODE BUFF" = 1) AND ("MODE SELECTION DB"."UF PLC_1 PROCESS BUFF" = 260) AND "INPUT MAPPING DB"."ABFV 202 FEED BACK CLOSE" THEN
       "MODE SELECTION DB"."UF PLC_1 PROCESS BUFF" := 265;
   END_IF;
END_REGION

REGION Network 59: 270
   RUNG wire#powerrail
      { S7_Templates := "SrcType := Int" } EQ_Contact(in1 := "MODE SELECTION DB"."UF PLC_1 MODE BUFF", in2 := 1)
      { S7_Templates := "SrcType := Int" } EQ_Contact(in1 := "MODE SELECTION DB"."UF PLC_1 PROCESS BUFF", in2 := 265)
      Move(in := 270, out1 => "MODE SELECTION DB"."UF PLC_1 PROCESS BUFF")
   END_RUNG
   // the same network as SCL:
   IF ("MODE SELECTION DB"."UF PLC_1 MODE BUFF" = 1) AND ("MODE SELECTION DB"."UF PLC_1 PROCESS BUFF" = 265) THEN
       "MODE SELECTION DB"."UF PLC_1 PROCESS BUFF" := 270;
   END_IF;
END_REGION

REGION Network 61: ABFV 201 OPEN FB
   RUNG wire#powerrail
      { S7_Templates := "SrcType := Int" } EQ_Contact(in1 := "MODE SELECTION DB"."UF PLC_1 MODE BUFF", in2 := 1)
      { S7_Templates := "SrcType := Int" } EQ_Contact(in1 := "MODE SELECTION DB"."UF PLC_1 PROCESS BUFF", in2 := 270)
      Contact( "INPUT MAPPING DB"."ABFV 201 FEED BACK OPEN" )
      Move(in := 275, out1 => "MODE SELECTION DB"."UF PLC_1 PROCESS BUFF")
   END_RUNG
   // the same network as SCL:
   IF ("MODE SELECTION DB"."UF PLC_1 MODE BUFF" = 1) AND ("MODE SELECTION DB"."UF PLC_1 PROCESS BUFF" = 270) AND "INPUT MAPPING DB"."ABFV 201 FEED BACK OPEN" THEN
       "MODE SELECTION DB"."UF PLC_1 PROCESS BUFF" := 275;
   END_IF;
END_REGION

REGION Network 62: ABFV 203 OPEN FB
   RUNG wire#powerrail
      { S7_Templates := "SrcType := Int" } EQ_Contact(in1 := "MODE SELECTION DB"."UF PLC_1 MODE BUFF", in2 := 1)
      { S7_Templates := "SrcType := Int" } EQ_Contact(in1 := "MODE SELECTION DB"."UF PLC_1 PROCESS BUFF", in2 := 275)
      Contact( "INPUT MAPPING DB"."ABFV 203 FEED BACK OPEN" )
      Move(in := 280, out1 => "MODE SELECTION DB"."UF PLC_1 PROCESS BUFF")
   END_RUNG
   // the same network as SCL:
   IF ("MODE SELECTION DB"."UF PLC_1 MODE BUFF" = 1) AND ("MODE SELECTION DB"."UF PLC_1 PROCESS BUFF" = 275) AND "INPUT MAPPING DB"."ABFV 203 FEED BACK OPEN" THEN
       "MODE SELECTION DB"."UF PLC_1 PROCESS BUFF" := 280;
   END_IF;
END_REGION

REGION Network 63: ABFV 206 OPEN FB
   RUNG wire#powerrail
      { S7_Templates := "SrcType := Int" } EQ_Contact(in1 := "MODE SELECTION DB"."UF PLC_1 MODE BUFF", in2 := 1)
      { S7_Templates := "SrcType := Int" } EQ_Contact(in1 := "MODE SELECTION DB"."UF PLC_1 PROCESS BUFF", in2 := 280)
      Contact( "INPUT MAPPING DB"."ABFV 206 FEED BACK OPEN" )
      { S7_Templates := "time_type := Time" } "IEC_Timer_0_DB_102".TON(pt := T#5S, et =>)
      Move(in := 285, out1 => "MODE SELECTION DB"."UF PLC_1 PROCESS BUFF")
   END_RUNG
   // the same network as SCL:
   "IEC_Timer_0_DB_102".TON(IN := ("MODE SELECTION DB"."UF PLC_1 MODE BUFF" = 1) AND ("MODE SELECTION DB"."UF PLC_1 PROCESS BUFF" = 280) AND "INPUT MAPPING DB"."ABFV 206 FEED BACK OPEN",
                           PT := T#5S);
   IF "IEC_Timer_0_DB_102".Q THEN "MODE SELECTION DB"."UF PLC_1 PROCESS BUFF" := 285; END_IF;
END_REGION

REGION Network 64: FORWARD FLUSH_2
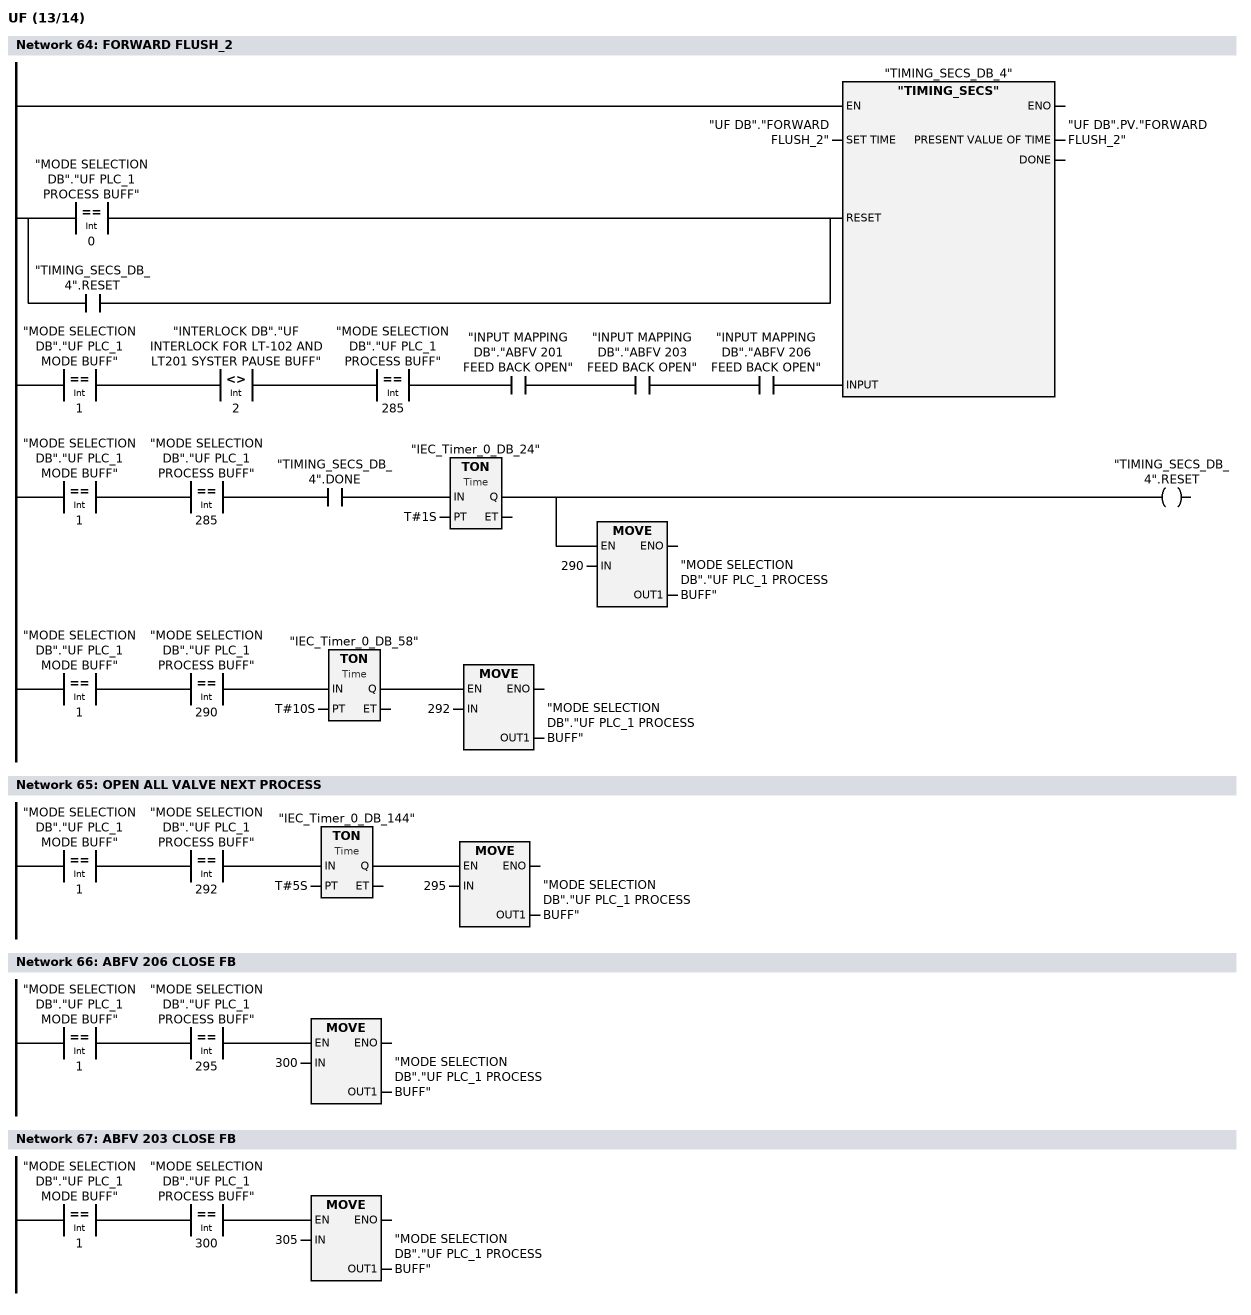
   RUNG wire#powerrail
      "TIMING_SECS_DB_4"(RESET := wire#w1, INPUT := wire#w2, "SET TIME" := "UF DB"."FORWARD FLUSH_2", "PRESENT VALUE OF TIME" => "UF DB".PV."FORWARD FLUSH_2", DONE =>)
   END_RUNG
   RUNG wire#powerrail
      { S7_Templates := "SrcType := Int" } EQ_Contact(in1 := "MODE SELECTION DB"."UF PLC_1 PROCESS BUFF", in2 := 0)
   END_RUNG wire#w1
   RUNG wire#powerrail
      Contact( "TIMING_SECS_DB_4".RESET )
   END_RUNG wire#w1
   RUNG wire#powerrail
      { S7_Templates := "SrcType := Int" } EQ_Contact(in1 := "MODE SELECTION DB"."UF PLC_1 MODE BUFF", in2 := 1)
      { S7_Templates := "SrcType := Int" } NE_Contact(in1 := "INTERLOCK DB"."UF INTERLOCK FOR LT-102 AND LT201 SYSTER PAUSE BUFF", in2 := 2)
      { S7_Templates := "SrcType := Int" } EQ_Contact(in1 := "MODE SELECTION DB"."UF PLC_1 PROCESS BUFF", in2 := 285)
      Contact( "INPUT MAPPING DB"."ABFV 201 FEED BACK OPEN" )
      Contact( "INPUT MAPPING DB"."ABFV 203 FEED BACK OPEN" )
      Contact( "INPUT MAPPING DB"."ABFV 206 FEED BACK OPEN" )
   END_RUNG wire#w2
   RUNG wire#powerrail
      { S7_Templates := "SrcType := Int" } EQ_Contact(in1 := "MODE SELECTION DB"."UF PLC_1 MODE BUFF", in2 := 1)
      { S7_Templates := "SrcType := Int" } EQ_Contact(in1 := "MODE SELECTION DB"."UF PLC_1 PROCESS BUFF", in2 := 285)
      Contact( "TIMING_SECS_DB_4".DONE )
      { S7_Templates := "time_type := Time" } "IEC_Timer_0_DB_24".TON(pt := T#1S, et =>)
      wire#w3
      Coil( "TIMING_SECS_DB_4".RESET )
   END_RUNG
   RUNG wire#w3
      Move(in := 290, out1 => "MODE SELECTION DB"."UF PLC_1 PROCESS BUFF")
   END_RUNG
   RUNG wire#powerrail
      { S7_Templates := "SrcType := Int" } EQ_Contact(in1 := "MODE SELECTION DB"."UF PLC_1 MODE BUFF", in2 := 1)
      { S7_Templates := "SrcType := Int" } EQ_Contact(in1 := "MODE SELECTION DB"."UF PLC_1 PROCESS BUFF", in2 := 290)
      { S7_Templates := "time_type := Time" } "IEC_Timer_0_DB_58".TON(pt := T#10S, et =>)
      Move(in := 292, out1 => "MODE SELECTION DB"."UF PLC_1 PROCESS BUFF")
   END_RUNG
   // the same network as SCL:
   "TIMING_SECS_DB_4"("SET TIME" := "UF DB"."FORWARD FLUSH_2",   // "TIMING_SECS"
                      RESET := ("MODE SELECTION DB"."UF PLC_1 PROCESS BUFF" = 0) OR "TIMING_SECS_DB_4".RESET,
                      INPUT := ("MODE SELECTION DB"."UF PLC_1 MODE BUFF" = 1) AND ("INTERLOCK DB"."UF INTERLOCK FOR LT-102 AND LT201 SYSTER PAUSE BUFF" <> 2) AND ("MODE SELECTION DB"."UF PLC_1 PROCESS BUFF" = 285) AND "INPUT MAPPING DB"."ABFV 201 FEED BACK OPEN" AND "INPUT MAPPING DB"."ABFV 203 FEED BACK OPEN" AND "INPUT MAPPING DB"."ABFV 206 FEED BACK OPEN",
                      "PRESENT VALUE OF TIME" => "UF DB".PV."FORWARD FLUSH_2");
   "IEC_Timer_0_DB_24".TON(IN := ("MODE SELECTION DB"."UF PLC_1 MODE BUFF" = 1) AND ("MODE SELECTION DB"."UF PLC_1 PROCESS BUFF" = 285) AND "TIMING_SECS_DB_4".DONE,
                           PT := T#1S);
   "TIMING_SECS_DB_4".RESET := "IEC_Timer_0_DB_24".Q;
   IF "IEC_Timer_0_DB_24".Q THEN "MODE SELECTION DB"."UF PLC_1 PROCESS BUFF" := 290; END_IF;
   "IEC_Timer_0_DB_58".TON(IN := ("MODE SELECTION DB"."UF PLC_1 MODE BUFF" = 1) AND ("MODE SELECTION DB"."UF PLC_1 PROCESS BUFF" = 290),
                           PT := T#10S);
   IF "IEC_Timer_0_DB_58".Q THEN "MODE SELECTION DB"."UF PLC_1 PROCESS BUFF" := 292; END_IF;
END_REGION

REGION Network 65: OPEN ALL VALVE NEXT PROCESS
   RUNG wire#powerrail
      { S7_Templates := "SrcType := Int" } EQ_Contact(in1 := "MODE SELECTION DB"."UF PLC_1 MODE BUFF", in2 := 1)
      { S7_Templates := "SrcType := Int" } EQ_Contact(in1 := "MODE SELECTION DB"."UF PLC_1 PROCESS BUFF", in2 := 292)
      { S7_Templates := "time_type := Time" } "IEC_Timer_0_DB_144".TON(pt := T#5S, et =>)
      Move(in := 295, out1 => "MODE SELECTION DB"."UF PLC_1 PROCESS BUFF")
   END_RUNG
   // the same network as SCL:
   "IEC_Timer_0_DB_144".TON(IN := ("MODE SELECTION DB"."UF PLC_1 MODE BUFF" = 1) AND ("MODE SELECTION DB"."UF PLC_1 PROCESS BUFF" = 292),
                           PT := T#5S);
   IF "IEC_Timer_0_DB_144".Q THEN "MODE SELECTION DB"."UF PLC_1 PROCESS BUFF" := 295; END_IF;
END_REGION

REGION Network 66: ABFV 206 CLOSE FB
   RUNG wire#powerrail
      { S7_Templates := "SrcType := Int" } EQ_Contact(in1 := "MODE SELECTION DB"."UF PLC_1 MODE BUFF", in2 := 1)
      { S7_Templates := "SrcType := Int" } EQ_Contact(in1 := "MODE SELECTION DB"."UF PLC_1 PROCESS BUFF", in2 := 295)
      Move(in := 300, out1 => "MODE SELECTION DB"."UF PLC_1 PROCESS BUFF")
   END_RUNG
   // the same network as SCL:
   IF ("MODE SELECTION DB"."UF PLC_1 MODE BUFF" = 1) AND ("MODE SELECTION DB"."UF PLC_1 PROCESS BUFF" = 295) THEN
       "MODE SELECTION DB"."UF PLC_1 PROCESS BUFF" := 300;
   END_IF;
END_REGION

REGION Network 67: ABFV 203 CLOSE FB
   RUNG wire#powerrail
      { S7_Templates := "SrcType := Int" } EQ_Contact(in1 := "MODE SELECTION DB"."UF PLC_1 MODE BUFF", in2 := 1)
      { S7_Templates := "SrcType := Int" } EQ_Contact(in1 := "MODE SELECTION DB"."UF PLC_1 PROCESS BUFF", in2 := 300)
      Move(in := 305, out1 => "MODE SELECTION DB"."UF PLC_1 PROCESS BUFF")
   END_RUNG
   // the same network as SCL:
   IF ("MODE SELECTION DB"."UF PLC_1 MODE BUFF" = 1) AND ("MODE SELECTION DB"."UF PLC_1 PROCESS BUFF" = 300) THEN
       "MODE SELECTION DB"."UF PLC_1 PROCESS BUFF" := 305;
   END_IF;
END_REGION

REGION Network 68: ABFV 201 CLOSE FB
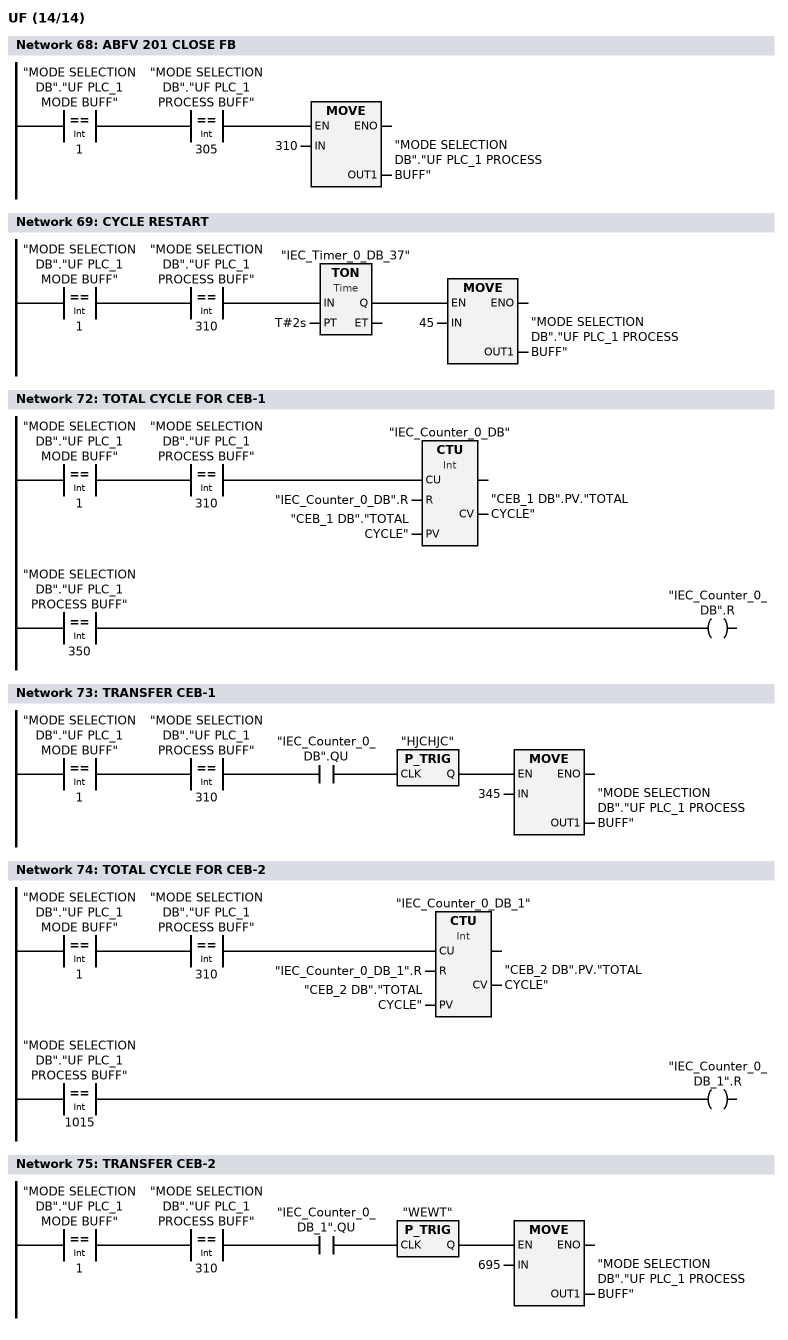
   RUNG wire#powerrail
      { S7_Templates := "SrcType := Int" } EQ_Contact(in1 := "MODE SELECTION DB"."UF PLC_1 MODE BUFF", in2 := 1)
      { S7_Templates := "SrcType := Int" } EQ_Contact(in1 := "MODE SELECTION DB"."UF PLC_1 PROCESS BUFF", in2 := 305)
      Move(in := 310, out1 => "MODE SELECTION DB"."UF PLC_1 PROCESS BUFF")
   END_RUNG
   // the same network as SCL:
   IF ("MODE SELECTION DB"."UF PLC_1 MODE BUFF" = 1) AND ("MODE SELECTION DB"."UF PLC_1 PROCESS BUFF" = 305) THEN
       "MODE SELECTION DB"."UF PLC_1 PROCESS BUFF" := 310;
   END_IF;
END_REGION

REGION Network 69: CYCLE RESTART
   RUNG wire#powerrail
      { S7_Templates := "SrcType := Int" } EQ_Contact(in1 := "MODE SELECTION DB"."UF PLC_1 MODE BUFF", in2 := 1)
      { S7_Templates := "SrcType := Int" } EQ_Contact(in1 := "MODE SELECTION DB"."UF PLC_1 PROCESS BUFF", in2 := 310)
      { S7_Templates := "time_type := Time" } "IEC_Timer_0_DB_37".TON(pt := T#2s, et =>)
      Move(in := 45, out1 => "MODE SELECTION DB"."UF PLC_1 PROCESS BUFF")
   END_RUNG
   // the same network as SCL:
   "IEC_Timer_0_DB_37".TON(IN := ("MODE SELECTION DB"."UF PLC_1 MODE BUFF" = 1) AND ("MODE SELECTION DB"."UF PLC_1 PROCESS BUFF" = 310),
                           PT := T#2s);
   IF "IEC_Timer_0_DB_37".Q THEN "MODE SELECTION DB"."UF PLC_1 PROCESS BUFF" := 45; END_IF;
END_REGION

REGION Network 72: TOTAL CYCLE FOR CEB-1
   RUNG wire#powerrail
      { S7_Templates := "SrcType := Int" } EQ_Contact(in1 := "MODE SELECTION DB"."UF PLC_1 MODE BUFF", in2 := 1)
      { S7_Templates := "SrcType := Int" } EQ_Contact(in1 := "MODE SELECTION DB"."UF PLC_1 PROCESS BUFF", in2 := 310)
      { S7_Templates := "value_type := Int" } "IEC_Counter_0_DB".CTU(r := "IEC_Counter_0_DB".R, pv := "CEB_1 DB"."TOTAL CYCLE", cv => "CEB_1 DB".PV."TOTAL CYCLE")
   END_RUNG
   RUNG wire#powerrail
      { S7_Templates := "SrcType := Int" } EQ_Contact(in1 := "MODE SELECTION DB"."UF PLC_1 PROCESS BUFF", in2 := 350)
      Coil( "IEC_Counter_0_DB".R )
   END_RUNG
   // the same network as SCL:
   "IEC_Counter_0_DB".CTU(CU := ("MODE SELECTION DB"."UF PLC_1 MODE BUFF" = 1) AND ("MODE SELECTION DB"."UF PLC_1 PROCESS BUFF" = 310),
                          R := "IEC_Counter_0_DB".R,
                          PV := "CEB_1 DB"."TOTAL CYCLE",
                          CV => "CEB_1 DB".PV."TOTAL CYCLE");
   "IEC_Counter_0_DB".R := "MODE SELECTION DB"."UF PLC_1 PROCESS BUFF" = 350;
END_REGION

REGION Network 73: TRANSFER CEB-1
   RUNG wire#powerrail
      { S7_Templates := "SrcType := Int" } EQ_Contact(in1 := "MODE SELECTION DB"."UF PLC_1 MODE BUFF", in2 := 1)
      { S7_Templates := "SrcType := Int" } EQ_Contact(in1 := "MODE SELECTION DB"."UF PLC_1 PROCESS BUFF", in2 := 310)
      Contact( "IEC_Counter_0_DB".QU )
      P_Trig( "HJCHJC" )
      Move(in := 345, out1 => "MODE SELECTION DB"."UF PLC_1 PROCESS BUFF")
   END_RUNG
   // the same network as SCL:
   #_w1 := ("MODE SELECTION DB"."UF PLC_1 MODE BUFF" = 1) AND ("MODE SELECTION DB"."UF PLC_1 PROCESS BUFF" = 310) AND "IEC_Counter_0_DB".QU;
   #_w2 := #_w1 AND NOT "HJCHJC";   // rising edge
   "HJCHJC" := #_w1;
   IF #_w2 THEN "MODE SELECTION DB"."UF PLC_1 PROCESS BUFF" := 345; END_IF;
END_REGION

REGION Network 74: TOTAL CYCLE FOR CEB-2
   RUNG wire#powerrail
      { S7_Templates := "SrcType := Int" } EQ_Contact(in1 := "MODE SELECTION DB"."UF PLC_1 MODE BUFF", in2 := 1)
      { S7_Templates := "SrcType := Int" } EQ_Contact(in1 := "MODE SELECTION DB"."UF PLC_1 PROCESS BUFF", in2 := 310)
      { S7_Templates := "value_type := Int" } "IEC_Counter_0_DB_1".CTU(r := "IEC_Counter_0_DB_1".R, pv := "CEB_2 DB"."TOTAL CYCLE", cv => "CEB_2 DB".PV."TOTAL CYCLE")
   END_RUNG
   RUNG wire#powerrail
      { S7_Templates := "SrcType := Int" } EQ_Contact(in1 := "MODE SELECTION DB"."UF PLC_1 PROCESS BUFF", in2 := 1015)
      Coil( "IEC_Counter_0_DB_1".R )
   END_RUNG
   // the same network as SCL:
   "IEC_Counter_0_DB_1".CTU(CU := ("MODE SELECTION DB"."UF PLC_1 MODE BUFF" = 1) AND ("MODE SELECTION DB"."UF PLC_1 PROCESS BUFF" = 310),
                           R := "IEC_Counter_0_DB_1".R,
                           PV := "CEB_2 DB"."TOTAL CYCLE",
                           CV => "CEB_2 DB".PV."TOTAL CYCLE");
   "IEC_Counter_0_DB_1".R := "MODE SELECTION DB"."UF PLC_1 PROCESS BUFF" = 1015;
END_REGION

REGION Network 75: TRANSFER CEB-2
   RUNG wire#powerrail
      { S7_Templates := "SrcType := Int" } EQ_Contact(in1 := "MODE SELECTION DB"."UF PLC_1 MODE BUFF", in2 := 1)
      { S7_Templates := "SrcType := Int" } EQ_Contact(in1 := "MODE SELECTION DB"."UF PLC_1 PROCESS BUFF", in2 := 310)
      Contact( "IEC_Counter_0_DB_1".QU )
      P_Trig( "WEWT" )
      Move(in := 695, out1 => "MODE SELECTION DB"."UF PLC_1 PROCESS BUFF")
   END_RUNG
   // the same network as SCL:
   #_w1 := ("MODE SELECTION DB"."UF PLC_1 MODE BUFF" = 1) AND ("MODE SELECTION DB"."UF PLC_1 PROCESS BUFF" = 310) AND "IEC_Counter_0_DB_1".QU;
   #_w2 := #_w1 AND NOT "WEWT";   // rising edge
   "WEWT" := #_w1;
   IF #_w2 THEN "MODE SELECTION DB"."UF PLC_1 PROCESS BUFF" := 695; END_IF;
END_REGION
END_FUNCTION
